// SIMATIC STEP 7 (V5.x) project AEX52
// CPU: CPU
// station: P_ADR_BUS
// station: _S7H_BUSSYSTEM_CT
// station: Matériel
// station: API
// station: P_ADR_BUS
// station: Configuration
// station: MOP
// program: PROG
// program: SAFETY_V2
// program: S120_CU320_2_PN

SYMBOL_TABLE
"ITS0"	DB 1100	FB 1100	// ILOT : DB INSTANCE FB1100
"ITSZ1_AU_ES_FZ"	DB 1110	FB 1110	// Z1 : DB D'INSTANCE DU FB 1110
"ITSZ1SOP"	DB 1111	FB 1111	// Z1 : DB D'INSTANCE DU FB 1111
"ITSZ1SOPR"	DB 1112	FB 1112	// Z1 : DB D'INSTANCE DU FB 1112
"ITSZ1VAR"	DB 1113	FB 1113	// Z1 : DB D'INSTANCE DU FB 1113
"TSM"	DB 1279	DB 1279	// STD - DB global pour la Tâche de Sécurité
"TSE_AMONT"	DB 1286	FB 1692	// STD - INSTANCE DB OF FB 1692 (F_SENDDP) SAFETY DATA SEND
"TSR_AMONT"	DB 1287	FB 1693	// STD - INSTANCE DB OF FB 1693 (F_RCVDP) SAFETY DATA RECEIVE
"TSE_AVAL"	DB 1288	FB 1692	// STD - INSTANCE DB OF FB 1692 (F_SENDDP) SAFETY DATA SEND
"TSR_AVAL"	DB 1289	FB 1693	// STD - INSTANCE DB OF FB 1693 (F_RCVDP) SAFETY DATA RECEIVE
"F_GLOBDB"	DB 1300	DB 1300	// F_: F_Global_Data Block
"F_TON"	FB 185	FB 185	// F_: Timer Switch On Delay
"F_TOF"	FB 186	FB 186	// F_: Timer Switch Off Delay
"TS0"	FB 1100	FB 1100	// ILOT: FB Gestion SAFETY ilot
"TSZ1_AU_ES_FZ"	FB 1110	FB 1110
"TSZ1_SOP"	FB 1111	FB 1111
"TSZ1_SOPR"	FB 1112	FB 1112
"TSZ1_VAR"	FB 1113	FB 1113
"F_SENDDP"	FB 1692	FB 1692	// F_: Send Data via PROFIBUS DP / PROFINET IO
"F_RCVDP"	FB 1693	FB 1693	// F_: Receive Data via PROFIBUS DP / PROFINET IO
"F_ACK_GL"	FB 1695	FB 1695	// Acquittement global de toutes les périphéries F d'un groupe d'exécution F
"BFS_BSEC1"	FB 1710	FB 1710
"BFS_BSECTR1"	FB 1711	FB 1711
"BFS_PORTE1"	FB 1712	FB 1712
"BFS_AIR1"	FB 1713	FB 1713
"BFS_CRM1"	FB 1714	FB 1714
"BFS_CR1"	FB 1715	FB 1715
"BFS_CAME_ROBOT1"	FB 1716	FB 1716
"BFS_MUT1"	FB 1717	FB 1717
"BFS_BIMA1"	FB 1721	FB 1721
"0_00_TSSAFETY"	FC 1100	FC 1100	// STD - FACILITY: EXECUTION F GROUP ASSOCIATE TO OB32 (NORMAL TASK)
"0_00_TSCYCLE"	FC 1101	FC 1101	// CALL OPERATOR NOT IN ZONE FB LINKED IN FACILITY
"P0OP1BAU1"	I 2.0	BOOL	// [P0SB1A.M08]: OPERATOR 1 EGS.CHANNEL 1 / BP ARRET D URGENCE OPERATEUR 1 (VOIE 1)
"P0OP2BAU1"	I 2.1	BOOL	// [P0SB1A.M08]: OPERATOR 2 EGS.CHANNEL 1 / BP ARRET D URGENCE OPERATEUR 2 (VOIE 1)
"P0OP3BAU1"	I 2.2	BOOL	// [P0SB1A.M08]: OPERATOR 3 EGS.CHANNEL 1 / BP ARRET D URGENCE OPERATEUR 3 (VOIE 1)
"P0OP4BAU1"	I 2.3	BOOL	// [P0SB1A.M08]: OPERATOR 4 EGS.CHANNEL 1 / BP ARRET D URGENCE OPERATEUR 4 (VOIE 1)
"P0OP1BAU2"	I 2.4	BOOL	// [P0SB1A.M08]: OPERATOR 1 EGS.CHANNEL 2 / BP ARRET D URGENCE OPERATEUR 1 (VOIE 2)
"P0OP2BAU2"	I 2.5	BOOL	// [P0SB1A.M08]: OPERATOR 2 EGS.CHANNEL 2 / BP ARRET D URGENCE OPERATEUR 2 (VOIE 2)
"P0OP3BAU2"	I 2.6	BOOL	// [P0SB1A.M08]: OPERATOR 3 EGS.CHANNEL 2 / BP ARRET D URGENCE OPERATEUR 3 (VOIE 2)
"P0OP4BAU2"	I 2.7	BOOL	// [P0SB1A.M08]: OPERATOR 4 EGS.CHANNEL 2 / BP ARRET D URGENCE OPERATEUR 4 (VOIE 2)
"P0OP1CPOP1"	I 3.0	BOOL	// [P0SB1A.M09]: LIGHT CURTAIN 1 OR LASER 1 (CH 1) / BARRIERE IMMAT OU SCRUTATEUR
"P0_FDI_RES11"	I 3.1	BOOL	// [P0SB1A.M09]: SPARE SAFE DIGITAL INPUT / RESERVE ENTREE DE SECURITE
"P0OP2CPOP1"	I 3.2	BOOL	// [P0SB1A.M09]: LIGHT CURTAIN 2 OR LASER 2 (CH 1) / BARRIERE IMMAT OU SCRUTATEUR
"P0_FDI_RES21"	I 3.3	BOOL	// [P0SB1A.M09]: SPARE SAFE DIGITAL INPUT / RESERVE ENTREE DE SECURITE
"P0OP1CPOP2"	I 3.4	BOOL	// [P0SB1A.M09]: LIGHT CURTAIN 1 OR LASER 1 (CH 2) / BARRIERE IMMAT OU SCRUTATEUR
"P0_FDI_RES12"	I 3.5	BOOL	// [P0SB1A.M09]: SPARE SAFE DIGITAL INPUT / RESERVE ENTREE DE SECURITE
"P0OP2CPOP2"	I 3.6	BOOL	// [P0SB1A.M09]: LIGHT CURTAIN 2 OR LASER 2 (CH 2) / BARRIERE IMMAT OU SCRUTATEUR
"P0_FDI_RES22"	I 3.7	BOOL	// [P0SB1A.M09]: SPARE SAFE DIGITAL INPUT / RESERVE ENTREE DE SECURITE
"P0OP3CPOP1"	I 4.0	BOOL	// [P0SB1A.M10]: LIGHT CURTAIN 3 (CHANNEL 1)  / BARRIERE IMMATERIELLE (VOIE 1)
"P0_FDI_RES31"	I 4.1	BOOL	// [P0SB1A.M10]: SPARE SAFE DIGITAL INPUT / RESERVE ENTREE DE SECURITE
"P0OP4CPOP1"	I 4.2	BOOL	// [P0SB1A.M10]: LIGHT CURTAIN 4 (CHANNEL 1)  / BARRIERE IMMATERIELLE (VOIE 1)
"P0_FDI_RES41"	I 4.3	BOOL	// [P0SB1A.M10]: SPARE SAFE DIGITAL INPUT / RESERVE ENTREE DE SECURITE
"P0OP3CPOP2"	I 4.4	BOOL	// [P0SB1A.M10]: LIGHT CURTAIN 3 (CHANNEL 2)  / BARRIERE IMMATERIELLE (VOIE 2)
"P0_FDI_RES32"	I 4.5	BOOL	// [P0SB1A.M10]: SPARE SAFE DIGITAL INPUT / RESERVE ENTREE DE SECURITE
"P0OP4CPOP2"	I 4.6	BOOL	// [P0SB1A.M10]: LIGHT CURTAIN 4 (CHANNEL 2)  / BARRIERE IMMATERIELLE (VOIE 2)
"P0_FDI_RES42"	I 4.7	BOOL	// [P0SB1A.M10]: SPARE SAFE DIGITAL INPUT / RESERVE ENTREE DE SECURITE
"Z1CCSC1"	I 10.0	BOOL	// (Z1ZB.M02): SAFETY COMMON CONTROL SC1
"Z1CCES"	I 10.1	BOOL	// (Z1ZB.M02): SAFETY COMMON CONTROL ES
"Z1CCFZ"	I 10.2	BOOL	// (Z1ZB.M02): SAFETY COMMON CONTROL FZ
"Z1CCSC4"	I 10.3	BOOL	// (Z1ZB.M02): SAFETY COMMON CONTROL SC4
"Z1CP7B"	I 11.0	BOOL	// (Z1ZB.M03): 7 BARS PRESSURE CONTROL
"Z1CRM"	I 11.1	BOOL	// (Z1ZB.M03): CHECK GROUND RELAY
"BAUI"	I 13.0	BOOL	// (Z1ZB.M07): FACILITY EMERGENCY STOP
"Z1BAU2"	I 13.1	BOOL	// (Z1ZB.M07): ZONE EMERGENCY STOP
"Z1SSZ"	I 13.2	BOOL	// (Z1ZB.M07): ZONE SAFETY SELECTOR
"Z1CPOP1"	I 19.0	BOOL	// (Z1ZB.M08): LIGHT CURTAIN 1
"Z1CPOP2"	I 19.1	BOOL	// (Z1ZB.M08): LIGHT CURTAIN 2
"Z1RB3CCB24Z"	I 60.4	BOOL	// (Z1RB3.M02): ELECTRICAL CIRCUIT BREAKER 24V (24Z)
"Z1RB3CCB24R"	I 60.5	BOOL	// (Z1RB3.M02): ELECTRICAL CIRCUIT BREAKER 24V (24R)
"Z1SPA1BMCY"	I 100.7	BOOL	// (Z1SPA1.I0): CYCLE START BUTTON
"Z1SPA1BDACY"	I 101.0	BOOL	// (Z1SPA1.I1): CYCLE STOP REQUEST BUTTON
"Z1SPA1SPES"	I 101.3	BOOL	// (Z1SPA1.I1): SWITCH ON / OFF GATE
"Z1SPA1SS"	I 103.7	BOOL	// (Z1SPA1.SI0): SAFETY SELECTOR
"Z1SPA1CFP"	I 104.0	BOOL	// (Z1SPA1.SI1): DOOR CLOSED CONTROL
"P0RBXCFRO_ES"	I 104.6	BOOL	// [P0RBX]: RB OUTPUT - FRO ES COMMON CHECK / CONTROLE FRO MISE EN SERVICE
"P0RBXCFRO_ZF1"	I 104.7	BOOL	// [P0RBX]: RB OUTPUT - FRO FZ1 COMMON CHECK / CONTROLE FRO FERMETURE ZONE 1
"P0RBXCFRO_ZF2"	I 105.0	BOOL	// [P0RBX]: RB OUTPUT - FRO FZ2 COMMON CHECK / CONTROLE FRO FERMETURE ZONE 2
"Z1SPA2BMCY"	I 110.7	BOOL	// (Z1SPA2.I0): CYCLE START BUTTON
"Z1SPA2BDACY"	I 111.0	BOOL	// (Z1SPA2.I1): CYCLE STOP REQUEST BUTTON
"Z1SPA2SPES"	I 111.3	BOOL	// (Z1SPA2.I1): SWITCH ON / OFF GATE
"Z1SPA2SS"	I 113.7	BOOL	// (Z1SPA2.SI0): SAFETY SELECTOR
"Z1SPA2CFP"	I 114.0	BOOL	// (Z1SPA2.SI1): DOOR CLOSED CONTROL
"ZZXCP7B"	I 201.0	BOOL	// [ZZXZB.M03]: CHECK EV 7 BARS
"ZZXCRM"	I 201.1	BOOL	// [ZZXZB.M03]: CHECK GROUND RELAY
"ZZXCCB400_1"	I 201.2	BOOL	// [ZZXZB.M03]: BREAKER CONTROL 400V (SDB1)
"ZZXCRO_11"	I 201.3	BOOL	// [ZZXZB.M03]: SAFETY CONTACTOR CONTROL 1 (SDB1)
"ZZXCRO_12"	I 201.4	BOOL	// [ZZXZB.M03]: SAFETY CONTACTOR CONTROL 2 (SDB1)
"ZZXCCB400_2"	I 201.5	BOOL	// [ZZXZB.M03]: BREAKER CONTROL 400V (SDB2)
"ZZXCRO_21"	I 201.6	BOOL	// [ZZXZB.M03]: SAFETY CONTACTOR CONTROL 1 (SDB2)
"ZZXCRO_22"	I 201.7	BOOL	// [ZZXZB.M03]: SAFETY CONTACTOR CONTROL 2 (SDB2)
"ZZXBAUI1"	I 202.0	BOOL	// [ZZXZB.M06]: EGS FACILITY (MOP/LOP) - CHANNEL 1
"ZZXBAU1"	I 202.1	BOOL	// [ZZXZB.M06]: EGS ZONE (SOP/DLOP) - CHANNEL 1
"ZZXSSZ1"	I 202.2	BOOL	// [ZZXZB.M06]: SAFETY ZONE SELECTOR - CHANNEL 1
"ZZXBAUI2"	I 202.4	BOOL	// [ZZXZB.M06]: EGS FACILITY (MOP/LOP) - CHANNEL 2
"ZZXBAU2"	I 202.5	BOOL	// [ZZXZB.M06]: EGS ZONE (SOP/DLOP) - CHANNEL 2
"ZZXSSZ2"	I 202.6	BOOL	// [ZZXZB.M06]: SAFETY ZONE SELECTOR - CHANNEL 2
"ZZXIFRO1"	I 213.0	BOOL	// [ZZXZB.M08]: FRO1 INTERNAL CHECK
"ZZXIFRO2"	I 214.0	BOOL	// [ZZXZB.M09]: FRO2 INTERNAL CHECK
"P0OPXBP11"	I 339.0	BOOL	// [P0SB1A.M09]: OPX T-STAND BUTTON 1 - CHANNEL 1 / BIMANUEL X BOUTON 1 (VOIE 1)
"P0OPXBP21"	I 339.1	BOOL	// [P0SB1A.M09]: OPX T-STAND BUTTON 2 - CHANNEL 1 / BIMANUEL X BOUTON 2 (VOIE 1)
"P0OPXBP12"	I 339.4	BOOL	// [P0SB1A.M09]: OPX T-STAND BUTTON 1 - CHANNEL 2 / BIMANUEL X BOUTON 1 (VOIE 2)
"P0OPXBP22"	I 339.5	BOOL	// [P0SB1A.M09]: OPX T-STAND BUTTON 2 - CHANNEL 2 / BIMANUEL X BOUTON 2 (VOIE 2)
"BA0"	M 0.0	BOOL	// FACILITY: BIT ALWAYS OFF
"BA1"	M 0.1	BOOL	// FACILITY: BIT ALWAYS ON
"BA1LIEN"	M 0.2	BOOL	// FACILITY: BIT ALWAYS ON (LINK IN THE PROGRAMMING NETWORK)
"SHUNT"	M 0.3	BOOL	// FACILITY: BIT  FOR BYPASS SOME FUNCTIONS DURING THE TEST
"PERSO"	M 0.4	BOOL	// NEED TO PERSONALIZE BY THE PROGRAMMER
"POUB"	M 0.5	BOOL	// BIT TRASH
"SYSFROID"	M 0.7	BOOL	// DETECTING COLD START PLC (OB102)
"DEF_MAJ"	M 10.0	BOOL	// FACILITY: MAJOR FAULT (SAFETY)
"IADF"	M 10.1	BOOL	// FACILITY: FAULT RESET INFORMATION (SAFETY)
"IR"	M 10.2	BOOL	// FACILITY: CONTROL ON INFORMATION (SAFETY)
"P0OP1CRSP0"	M 12.0	BOOL	// P0: SAFETY RESET CONDITION / CONDITION DE REARMEMENT SECURITE
"P0OP2CRSP0"	M 12.1	BOOL	// P0: SAFETY RESET CONDITION / CONDITION DE REARMEMENT SECURITE
"Z1DEF_MAJ"	M 100.0	BOOL	// ZONE 1: MAJOR FAULT (SAFETY)
"Z1IADF"	M 100.1	BOOL	// ZONE 1: FAULT RESET INFORMATION (SAFETY)
"Z1IR"	M 100.2	BOOL	// ZONE 1: CONTROL ON INFORMATION (SAFETY)
"Z1IAFJ"	M 100.3	BOOL	// ZONE 1: END OF PRODUCTION STOP INFORMATION (SAFETY)
"P0OPXCRSP0"	M 103.2	BOOL	// P0OPX: SAFETY RESET CONDITION / CONDITION DE REARMEMENT SECURITE
"ZZXDEF_MAJ"	M 200.0	BOOL	// ZONE ZX: MAJOR FAULT (SAFETY)
"ZZXIADF"	M 200.1	BOOL	// ZONE ZX: FAULT RESET INFORMATION (SAFETY)
"ZZXIR"	M 200.2	BOOL	// ZONE ZX: CONTROL ON INFORMATION (SAFETY)
"ZZXIAFJ"	M 200.3	BOOL	// ZONE ZX: END OF PRODUCTION STOP INFORMATION (SAFETY)
"P0IAVARR"	M 201.0	BOOL	// P0: INFORMATION INVERTER STOP / INFO ARRET IMMEDIAT VARIATEUR
"P0_AT_P0OPX"	M 204.0	BOOL	// P0: OPERATOR P0OPX WORK AUTORIZATION / AUTORISATION DE TRAVAIL OPERATEUR P0OPX
"P0_ET_P0OPX"	M 204.1	BOOL	// P0: OPERATOR P0OPX WORK RECORD / ENREGISTREMENT TRAVAIL OPERATEUR P0OPX
"Z1RCM"	Q 10.7	BOOL	// (Z1ZB.M05): CHECK GROUND RELAY
"Z1RSC1"	Q 25.0	BOOL	// (Z1ZB.M09): SAFETY COMMON RELAY SC1
"Z1RES"	Q 25.1	BOOL	// (Z1ZB.M09): SAFETY COMMON RELAY ES
"Z1RFZ"	Q 25.2	BOOL	// (Z1ZB.M09): SAFETY COMMON RELAY FZ
"Z1RSC4"	Q 25.3	BOOL	// (Z1ZB.M09): SAFETY COMMON RELAY SC4
"DPRD_DAT"	SFC 14	SFC 14	// Read Consistent Data of a Standard DP Slave
"DPWR_DAT"	SFC 15	SFC 15	// Write Consistent Data to a Standard DP Slave
"STP"	SFC 46	SFC 46	// Change the CPU to STOP
END_SYMBOL_TABLE

// FB 185: know-how protected block, not included

// FB 186: know-how protected block, not included

FUNCTION_BLOCK "TS0"	// FB 1100
VERSION : 0.3
VAR
  ACK_GLB : FB 1695;	//FACILITY: GLOBAL FAULT RESET FOR SAFETY MODULE/AQUIT GENERAL DEF MATERIEL SAFET
  Z1CRM : FB 1714;	//Z1: GROUND RELAY CHECK / CONTROLE RELAI DE MASSE
END_VAR
BEGIN
// body was compiled from another editor; compiled code not shown
END_FUNCTION_BLOCK

FUNCTION_BLOCK "TSZ1_AU_ES_FZ"	// FB 1110
VERSION : 0.3
VAR
  Z1AU : FB 1710;	//Z1: EMERGENCY STOP RELAY CONTROL / GESTION BOUCLE DE SECURITE AU
  Z1ES : FB 1710;	//Z1: POWER ON RELAY CONTROL / GESTION RELAY MISE EN SERVICE
  Z1FZ : FB 1710;	//Z1: CLOSED ZONE SAFETY LOOP MANAGEMENT / GESTION BOUCLE DE SECURITE FZ
  Z1AIR : FB 1713;	//Z1: PRESSURIZING VALVE CONTROL / GESTION ELECTROVANNE DE MISE EN AIR
  Z1PORTE1 : FB 1712;	//Z1: DOOR 1 CONTROL / GESTION PORTE 1
  Z1PORTE2 : FB 1712;	//Z1: DOOR 2 CONTROL / GESTION PORTE 2
END_VAR
VAR_TEMP
  X1IBFF : BOOL ;	//AUX1 SAFETY CIRCUIT CORRECT WORKING INFORMATION / AUX BON FONCTIONNEMENT FILERI
  X2IBFF : BOOL ;	//AUX2 SAFETY CIRCUIT CORRECT WORKING INFORMATION / AUX BON FONCTIONNEMENT FILERI
  X3IBFF : BOOL ;	//AUX3 SAFETY CIRCUIT CORRECT WORKING INFORMATION / AUX BON FONCTIONNEMENT FILERI
  X1AUCAR : BOOL ;	//AUX1 CONDITIONS WITH RESET EMERGENCY STOP / AUX CONDITION AVEC REARMEMENT AU
  X2AUCAR : BOOL ;	//AUX2 CONDITIONS WITH RESET EMERGENCY STOP / AUX CONDITION AVEC REARMEMENT AU
  X1ESCAR : BOOL ;	//AUX1 CONDITIONS WITH RESET POWER ON / AUX1 CONDITIONS AVEC REARMEMENT EN SERVIC
  X2ESCAR : BOOL ;	//AUX2 CONDITIONS WITH RESET POWER ON / AUX2 CONDITIONS AVEC REARMEMENT EN SERVIC
END_VAR
BEGIN
// body was compiled from another editor; compiled code not shown
END_FUNCTION_BLOCK

FUNCTION_BLOCK "TSZ1_SOP"	// FB 1111
TITLE = POWER ON RELAY CONTROL
VERSION : 0.2
VAR
  C0SOP : FB 1710;
  F0SOP : FB 1710;
  G0SOP : FB 1710;
  P0SOP : FB 1710;
  P01SOP : FB 1710;
  P01SOP_Secu : BOOL ;	//Activation boucle de sécurité opérateur
  P02SOP : FB 1710;
  P02SOP_Secu : BOOL ;	//Activation boucle de sécurité opérateur
  F1BIMA : FB 1719;
  F2BIMA : FB 1719;
  F3BIMA : FB 1719;
END_VAR
VAR_TEMP
  C0SOP_Car : BOOL ;
  C0SOP_Csr : BOOL ;
  G0SOP_Car : BOOL ;
  G0SOP_Csr : BOOL ;
  P0SOP_Car : BOOL ;
  P0SOP_Csr : BOOL ;
  P01SOP_Car : BOOL ;
  P01SOP_Csr : BOOL ;
  P02SOP_Car : BOOL ;
  P02SOP_Csr : BOOL ;
  F0SOP_Car : BOOL ;
  F0SOP_Csr : BOOL ;
  C0SOP_csecu0 : BOOL ;
  C0SOP_csecu1 : BOOL ;
  F0SOP_csecu0 : BOOL ;
  F0SOP_csecu1 : BOOL ;
  G0SOP_csecu0 : BOOL ;
  G0SOP_csecu1 : BOOL ;
  P0SOP_csecu0 : BOOL ;
  P0SOP_csecu1 : BOOL ;
  P01SOP_csecu0 : BOOL ;
  P01SOP_csecu1 : BOOL ;
  P02SOP_csecu0 : BOOL ;
  P02SOP_csecu1 : BOOL ;
END_VAR
BEGIN
// body was compiled from another editor; compiled code not shown
END_FUNCTION_BLOCK

FUNCTION_BLOCK "TSZ1_SOPR"	// FB 1112
TITLE = CLOSED ZONE ELECTRICAL COMMON MANAGEMENT (FZ)
//GESTION DU COMMUN ELECTRIQUE : FERMETURE ZONE (FZ)
VERSION : 0.2
VAR
  R1CAME : FB 1716;
  R1SOPR : FB 1710;
END_VAR
VAR_TEMP
  R1SOPR_Car : BOOL ;	//R1 Conditions avec réarmement
  R1SOPR_Csr : BOOL ;	//R1 Conditions sans réarmement
  R1SOPR_csecu0 : BOOL ;
  R1SOPR_csecu1 : BOOL ;
END_VAR
BEGIN
// body was compiled from another editor; compiled code not shown
END_FUNCTION_BLOCK

FUNCTION_BLOCK "TSZ1_VAR"	// FB 1113
VERSION : 0.2
VAR
  Z1FZTR : FB 1711;	//Z1: CLOSED ZONE TEMPO SAFETY LOOP MANAGEMENT / GESTION BOUCLE SECURITE FZTR
END_VAR
BEGIN
// body was compiled from another editor; compiled code not shown
END_FUNCTION_BLOCK

// FB 1692: know-how protected block, not included

// FB 1693: know-how protected block, not included

// FB 1695: know-how protected block, not included

FUNCTION_BLOCK "BFS_BSEC1"	// FB 1710
//**********************************************************************
//*                             BFS_BSEC1                               *
//**********************************************************************
//(in english further below)
//DESCRIPTION: 
//************ 
//Le FB1710 "BFS_BSEC1" est un relais de securite logiciel programme en Step7 + 
//Distributed Safety pour assurer la surete de fonctionnement d'une boucle de 
//securite geree par automate Simatic Failsafe.
//C'est une evolution de la BFS_BSEC pour le Scube Safety V2
//
//Son role est 
//"De piloter une sortie F-DO ou PME-F, sur laquelle est cablee en fonction 
//du besoin process, un contacteur pour les energies de puissance 
//securisees et/ou un relais pour les communs de commande 24V et/ou une 
//electrovanne pour les energies de puissance pneumatiques. 
//"De controler la coherence entre le pilotage et l'etat des retours
//"De mettre a disposition du programme standard un commun de securite " 
//soft " pour conditionner le pilotage des sorties automates des mouvements a la 
//presence effective des communs de commande 24V et/ou des energies de puissance 
//et aussi pour conditionner les communs en aval (effet cascade)
//"D'avertir du mauvais fonctionnement de la boucle de securite (Alarme : 
//pas de retour alors que la sortie est pilotee, Defaut : retour present alors 
//que la sortie n'est pas pilotee)
//
//Le FB prend en compte les informations necessaires a la securisation de la 
//boucle de securite concernee.
//Il renseigne sur l'etat de defaillance de la fonction de securite.
//
//Les blocs associes pour le diagnostic via IHMP+ sont :
//BF_IHMCR1 pour les fonctions AU, ES, ZF et toute autre utilisation du 
//BFS_BSEC1 par exemple SOP …
//Le bloc BFS_BSEC1 peut egalement etre utilise pour la gestion du RL (Relais de 
//ligne) des fonctions variateurs Scube (Attention dans ce cas le diagnostic, pour 
//IHMP+, est realise par la BF associee a la fonction variateur)
//
//
//*************************English Information*******************************
//Description
//***********
//The FB1710 "BFS_BSEC1" is a software safety relay in Step 7 + Distributed 
//Safety to ensure the dependability of a safety loop managed by a Simatic 
//Failsafe PLC.
//It's an evolution of the BFS_BSEC with the Safety Scube V2.
//
//It serves: 
//"to control an F-DO or PME-F output, to which a contactor for the 
//safe power supplies and/or an relay for the safe commons 24V and/or a solenoid 
//valve for the safe power pneumatic fluid is/are wired according to process 
//requirements.
//"to check the consistency between the control and the status of the 
//feedbacks
//"to make a "software" safe common 24 V available to the standard program, to 
//make the control of PLC movement outputs conditional on the effective presence 
//of 24V control commons and/or power supplies and also to make the downstream 
//commons 24 V conditional (daisy-chained effect)
//"to give the alert in the event of incorrect operation of the safety loop 
//(Alarm: no feedback although the output is controlled, Fault: feedback present 
//although the output is not controlled)
//
//The FB takes into account the Data required to secure the safety loop concerned.
//It gives details on the failure status of the safety function and updates the 
//data from lien_sec used in the standard program.
//
//The associated blocks for the diagnostics via IHMP+ are:
//BF_IHMCR1 for the functions AU, ES, ZF and any other use of BFS_BSEC1 for 
//example SOP …
//The block BFS_BSEC1 can also be used to manage the RL (Line relay)of the Scube 
//drive functions (Attention in this case the diagnosis, for IHMP+, is carried out 
//with the BF associated with the drive function. 
//
AUTHOR : SIEMENS
FAMILY : RENAULT
NAME : BSEC1
VERSION : 1.0
VAR_INPUT
  Ibff : BOOL ;	//Safety circuit correct working info./Information bon fonctionnement filerie
  Car : BOOL ;	//Conditions with control on/Conditions avec rearmement
  Csr : BOOL ;	//Conditions without control on/Conditions sans rearmement
  CSecu0 : BOOL ;	//Feedbacks check without control/Controle Retours sans pilotage
  CSecu1 : BOOL ;	//Feedbacks check with control/Controle Retours avec Pilotage
  Iadf : BOOL ;	//Fault reset/Annulation defaut
  Ir : BOOL ;	//Function control on/Rearmement fonction
END_VAR
VAR_OUTPUT
  DO_F : BOOL ;	//F-DO output control/Commande sortie F-DO
  Secu : BOOL ;	//Similar with DO-F/Identique a DO_F
  Secu_OK : BOOL ;	//Safety loop correct/Boucle de securite valide
  Def : BOOL ;	//Discrepancy fault in the deactivation/Defaut de discordance a la desactivation
END_VAR
VAR
  x : BOOL  := TRUE;	//Bit of instance location/Bit de localisation de l'instance
  IHMDef : BOOL ;	//Discrepancy fault in the deactivation/Defaut de discordance a la desactivation
  IHMAla : BOOL ;	//Discrepancy fault in the activation/Def de discordance a l'activation (Ala)
  xSecu : BOOL ;	//Auxiliary bit/Bit auxiliaire
  M_ala : BOOL ;	//Alarm memory/Memoire alarme
  M_ar : BOOL ;	//Car memory (cond with Ctrl On)/Memoire car
  xIr : BOOL ;	//Auxiliary bit control on/Bit auxiliaire rearmement
  TON_Disc : FB 185;	//Discrepancy detection timer/Tempo de detection discordance
END_VAR
VAR_TEMP
  FP_Ir : BOOL ;	//Rising edge bit Ir (Control on information)/Bit front montant Ir
END_VAR
BEGIN
// body was compiled from another editor; compiled code not shown
END_FUNCTION_BLOCK

FUNCTION_BLOCK "BFS_BSECTR1"	// FB 1711
//**********************************************************************
//*                            BFS_BSECTR1                              *
//**********************************************************************
//(in english further below)
//DESCRIPTION: 
//************ 
//Le FB1711 "BFS_BSECTR1" est un relais de securite logiciel temporise a la 
//retombee programme en Step7 + Distributed Safety pour assurer la surete de 
//fonctionnement d'une boucle de securite gere par automate Simatic Failsafe.
//C'est une evolution de la BFS_BSECTR pour le Scube Safety V2
//
//Son role est 
//"De piloter une sortie F-DO ou PME-F temporise a la retombee, sur 
//laquelle est cablee en fonction du besoin process, un contacteur
//pour les energies de puissance securisees et/ou un relais pour 
//les communs de commande 24V securises.
//"De controler la coherence entre le pilotage et l'etat des retours
//"De mettre a disposition du programme standard un commun de securite " 
//soft " pour conditionner le pilotage des sorties automates des mouvements a la 
//presence effective des communs de commande 24V et/ou des energies de puissance
//"D'avertir du mauvais fonctionnement de la boucle de securite (Alarme : 
//pas de retour alors que la sortie est pilotee, Defaut : retour present alors 
//que la sortie n'est pas pilotee)
//
//Le FB prend en compte les informations necessaires a la securisation de la 
//boucle de securite concernee.
//
//Il renseigne sur l'etat de defaillance de la fonction de securite. 
//
//Les blocs associes pour le diagnostic via IHMP+ sont :
//BF_IHMCR1 pour la fonction ESTR ou toutes les autres utilisation du 
//BFS_BSECTR1
//
//*************************English Information*******************************
//Description
//***********
//The FB1711 "BFS_BSECTR" is a software safety relay with a delay when 
//falling, programmed in Step 7 + Distributed Safety to ensure the dependability 
//of a safety loop managed by a Simatic Failsafe PLC.
//It's an evolution of the BFS_BSEC with the Safety Scube V2.
//
//It serves: 
//"to control an F-DO or PME-F output with a deactivation delay, to which a 
//contactor for the safe power supplies and/or a relay for the safe commons 24V 
//is/are wired according to process requirements.
//"to check the consistency between the control and the status of the feedbacks
//"to make a "software" safe common 24 V available to the standard program, to 
//make the control of PLC movement outputs conditional on the effective presence 
//of 24V control commons and/or power supplies. 
//"to give the alert in the event of incorrect operation of the safety loop 
//(Alarm: no feedback although the output is controlled, Fault: feedback present 
//although the output is not controlled)
//
//The FB takes account of the Data required to secure the safety loop concerned.
//It gives details on the failure status of the safety function.
//
//The associated blocks for the diagnostics via IHMP+ are:
//BF_IHMCR1 for the ESTR function or all other uses of BFS_BSECTR1 
//BF_FONC_VAR_S for the RL function of FONC_VAR
AUTHOR : SIEMENS
FAMILY : RENAULT
NAME : BSECTR1
VERSION : 1.0
VAR_INPUT
  DSecu : BOOL ;	//Safety dependence/Dependance securite
  Cci : BOOL ;	//Immediate cut-off conditions/Conditions coupure immediate
  CSecu0 : BOOL ;	//Feedbacks check without control/Controle Retours sans pilotage
  CSecu1 : BOOL ;	//Feedbacks check with control/Controle Retours avec Pilotage
  Iadf : BOOL ;	//Fault reset/Annulation defaut
  Ir : BOOL ;	//Function control on/Rearmement fonction
  Tps_secu : TIME ;	//Relay deactivating time(Max.=2s)/Temps de retombee du relais (Maxi 2s
END_VAR
VAR_OUTPUT
  DO_F : BOOL ;	//F-DO output control/Commande sortie F-DO
  Secu : BOOL ;	//Similar with DO-F/Identique à DO_F
  Secu_OK : BOOL ;	//Safety loop correct/Boucle de securite valide
  Def : BOOL ;	//Discrepancy fault in the deactivation/Défaut de discordance à la desactivation
END_VAR
VAR
  x : BOOL ;	//Bit of instance location/Bit de localisation de l'instance
  IHMDef : BOOL ;	//Discrepancy fault in the deactivation/Defaut de discordance a la desactivation
  IHMAla : BOOL ;	//Discrepancy fault in the activation/Def de discordance a l'activation (Ala)
  xSecu : BOOL ;	//Auxiliary bit/Bit auxiliaire
  M_ala : BOOL ;	//Alarm memory/Memoire alarme
  M_Cci : BOOL ;	//Cci memory / memoire Cci
  xIr : BOOL ;	//Auxiliary bit control on/Bit auxiliaire rearmement
  TON_Disc : FB 185;	//Discrepancy detection timer/Tempo de detection discordance
  TOFF_Max : FB 186;	//Timer of relay deactivation with 2s max./Tempo de retombee relais avec 2 s max
  TOFF_Secu : FB 186;	//Timer of relay deactivation/Tempo de retombee relais
END_VAR
VAR_TEMP
  FP_Ir : BOOL ;	//Rising edge bit Ir (Control on information)/Bit front montant Ir
END_VAR
BEGIN
// body was compiled from another editor; compiled code not shown
END_FUNCTION_BLOCK

FUNCTION_BLOCK "BFS_PORTE1"	// FB 1712
//**********************************************************************
//*                             BFS_PORTE1                              *
//**********************************************************************
//(in english further below)
//DESCRIPTION: 
//************ 
//Le FB1712 "BFS_PORTE1" est un relais de securite logiciel programme en Step7 + 
//Distributed Safety.
//C'est une evolution de la BFS_PORTE pour le Scube Safety V2
//
//Ce FB assure la gestion des composants associes a une porte d'acces Zone.
//Il fournit les conditions pour l'activation des boucles de securité ES et ZF.
//Il controle le respect de la procedure d'intervention dans la zone.
//Il controle le bon fonctionnement de la gache, desactivation de 
//l'information cfp a chaque ouverture d'un des deux commutateurs SS ou SPES.
//
//Le blocs associe pour le diagnostic via IHMP+ est:
//BF_IHMPORTE1
//
//*************************English Information*******************************
//Description
//***********
//The FB1712 "BFS_BSEC1" is a software safety relay in Step 7 + Distributed 
//Safety. 
//It's an evolution of the BFS_PORTE with the Safety Scube V2.
//
//This FB ensures the management of components combined with a access gate into 
//an 
//area.
//It gives the conditions for the activation of safety loops ES and ZF. 
//It checks the respect of the intervention procedure in the area.
//It checks the correct working of the striker, deactivation of information cfp 
//in every opening of one of both switches SS or SPES.
//
//The associated block for the diagnostic via IHMP+ is:
//BF_IHMPORTE1 
AUTHOR : SIEMENS
FAMILY : RENAULT
NAME : PORTE1
VERSION : 1.0
VAR_INPUT
  Ss : BOOL ;	//Safety selector/Selecteur de Securite
  Cfp : BOOL ;	//Door closing check/Controle Fermeture Portillon
  Spes : BOOL ;	//Door enable selector/Selecteur Portillon En Service
  Iadf : BOOL ;	//Fault reset/Acquittement
END_VAR
VAR_OUTPUT
  ES_Car : BOOL ;	//Door validated for ES/Porte Ok pour ES
  FZ_Car : BOOL ;	//Door validated for FZ/Porte Ok pour FZ
END_VAR
VAR
  x : BOOL ;	//Bit of instance location/Bit de localisation de l'instance
  DPI : BOOL ;	//Maintenance procedure fault/Defaut procedure d'intervention
  DemOuv : BOOL ;	//Request for door opening/Demande ouvertrure porte
  XSel : BOOL ;	//Edge auxiliary/Auxilliaire de front
END_VAR
BEGIN
// body was compiled from another editor; compiled code not shown
END_FUNCTION_BLOCK

FUNCTION_BLOCK "BFS_AIR1"	// FB 1713
//**********************************************************************
//*                             BFS_AIR1                                *
//**********************************************************************
//(in english further below)
//DESCRIPTION: 
//************ 
//Le FB1713 assure la gestion d'un panneau pneumatique pour une zone. Il peut 
//piloter les electrovannes 7 bars de mise en pression progressive et de shunt de 
//mise en pression progressive.
//C'est une evolution de la BFS_BSECTR pour le Scube Safety V2
// 
//Attention ce pilotage peut egalement etre realise par la sortie securisee de la 
//boucle ES.
//Le FB genere des defauts en cas de dysfonctionnement (incoherence entre le 
//pilotage des electrovannes et le controle de pression pneumatique).
//Ce FB est prevu pour etre utilise avec un panneau classique, comportant les 
//commandes d'une electrovanne de mise en pression progressive et une 
//electrovanne de shunt de mise en pression progressive et un controle de 
//pression.
//Mais il peut egalement etre utilise pour un panneau comportant uniquement  les 
//commandes d'une electrovanne de ligne 7 bars et d'un controle de pression. Dans 
//ce cas, on utilisera la sortie EVMPP pour la commande de l'electrovanne.
//
//Le bloc associe pour le diagnostic via IHMP+ est :
//BF_IHMAIR1
//
//*************************English Information*******************************
//Description
//***********
//The FB1713 manages a zone's air panel. It can control the line solenoid valves 
//(7 Bar) of gradual pressurising and gradual pressurising shunt.
//It's an evolution of the BFS_AIR with the Safety Scube V2. 
//
//Note that this control can also be performed by the In Service loop secured 
//output.
//The FB generates faults if a malfunction occurs (discrepancy between the 
//solenoid valve controls and the air pressure check).
//This FB is designed to be used with a standard panel, including a gradual 
//pressurising solenoid valve, a gradual pressuring shunt solenoid valve and an 
//air pressure check.
//It can also be used for a panel that only has a line solenoid valve (7 bar) and 
//an air pressure check. In this case, we use the EVMPP output for the solenoid 
//valve control.
//
//The associated block for the diagnostic via IHMP+ is:
//BF_IHMAIR1
//
AUTHOR : SIEMENS
FAMILY : RENAULT
NAME : AIR1
VERSION : 1.0
VAR_INPUT
  DSecu : BOOL ;	//Safety dependence/Dependance securite
  Cpa7B : BOOL ;	//Air pressure 7 bars check/Controle Pression Air 7 bars
  Iadf : BOOL ;	//Fault reset/Annulation defaut
  Ir : BOOL ;	//Function control on/Rearmement fonction
  Vptmpp : TIME ;	//Setting value of gradual pressure timer/Val.Paramet.Tempo Mise en Pres. Progr.
END_VAR
VAR_OUTPUT
  EvMPP : BOOL ;	//EV Gradual pressurising valve/EV mise en pression progressive
  ShEvMPP : BOOL ;	//Shunt EV Gradual pressurising valve/Shunt EV mise en pression progressive
  Secu_Ok : BOOL ;	//Pressure air OK/Air Ok
  Def : BOOL ;	//Air fault/Defaut air
END_VAR
VAR
  x : BOOL ;	//Bit of instance location/Bit de localisation de l'instance
  IHMAla : BOOL ;	//Air pressure alarm/Alarme air
  IHMDef : BOOL ;	//Air pressure fault / Defaut Air
  MppT : BOOL ;	//Gradual pressurising time elapsed/Mise en Pression progressive terminee
  Mcp7b : BOOL ;	//Air pressure check memory/Memoire controle pression air
  M_ala : BOOL ;	//Alarm memory/ Memoire alarme
  xIr : BOOL ;	//Auxiliary bit control on/Bit auxiliaire rearmement
  TON_Mpp : FB 185;	//Gradual pressurising timer/Tempo mise en pression progressive
  TON_Disc : FB 185;	//Air fault detection timer/Tempo detection defaut air
END_VAR
VAR_TEMP
  FP_Ir : BOOL ;	//Rising edge bit Ir (Control on information)/Bit front montant Ir
END_VAR
BEGIN
// body was compiled from another editor; compiled code not shown
END_FUNCTION_BLOCK

FUNCTION_BLOCK "BFS_CRM1"	// FB 1714
//**********************************************************************
//*                               BFS_CRM1                              *
//**********************************************************************
//(in english further below)
//DESCRIPTION: 
//************ 
//Le FB1714 "BFS_CRM1" est un relais de securite logiciel programme en Step7 + 
//Distributed Safety.
//Il controle l'etat du relais de controle de masse .
//C'est une evolution de la BFS_CRM pour le Scube Safety V2
//
//Il est a appeler autant de fois qu'il y a d'alimentation 24V.
//Le bloc associe pour le diagnostic via IHMP+ est :
//BF_IHMCRM1
//
//*************************English Information*******************************
//Description
//***********
//The "BFS_CRM1" FB1714 is a software safety relay programmed in Step 7 + 
//Distributed Safety.
//It checks the status of the earthing check relay.
//It's an evolution of the BFS_CRM with the Safety Scube V2.
//
//It is to be integrated for each 24V control power supply.
//The associated block for the diagnostic via IHMP+ is:
//BF_IHMCRM1
AUTHOR : SIEMENS
FAMILY : RENAULT
NAME : CRM1
VERSION : 1.0
VAR_INPUT
  DSecu : BOOL ;	//Safety dependence/Dependance securite
  CSecu : BOOL ;	//Relay feedback information/Information de retour du relais
  Iadf : BOOL ;	//Fault reset/Annulation defaut
END_VAR
VAR_OUTPUT
  Def : BOOL ;	//CRM fault/Defaut CRM
END_VAR
VAR
  x : BOOL ;	//Bit of instance location/Bit de localisation de l'instance
  IHMDef : BOOL ;	//Fault in the deactivation/Defaut a la retombee
  IHMAla : BOOL ;	//Fault in the activation/Defaut a la montee
  xSecu : BOOL ;	//Auxiliary bit/Bit auxiliaire
  Ton_Rsecu : FB 185;	//Timer of discrepancy detection/Tempo de detection discordance
END_VAR
BEGIN
// body was compiled from another editor; compiled code not shown
END_FUNCTION_BLOCK

FUNCTION_BLOCK "BFS_CR1"	// FB 1715
//**********************************************************************
//*                               BFS_CR1                               *
//**********************************************************************
//(in english further below)
//DESCRIPTION: 
//************ 
//Le FB1715 "BFS_CR1" est un relais de securite logiciel programme en Step7 + 
//Distributed Safety.
//C'est une evolution de la BFS_CR pour le Scube Safety V2
//
//Il verifie la coherence entre la commande d'un relais et son etat. 
//
//Le bloc associe pour le diagnostic via IHMP+ est :
//BF_IHMCR1
//
//*************************English Information*******************************
//Description
//***********
//The "BFS_CR1" FB1715 is a software safety relay programmed in Step 7 + 
//Distributed Safety.
//It's an evolution of the BFS_CR with the Safety Scube V2.
//
//It checks the consistency between the relay control and its state.
//
//The associated block for the diagnostic via IHMP+ is:
//BF_IHMCR1
AUTHOR : SIEMENS
FAMILY : RENAULT
NAME : CR1
VERSION : 1.0
VAR_INPUT
  DSecu : BOOL ;	//Conditions with control on/Conditions avec rearmement
  CSecu0 : BOOL ;	//Feedbacks check without control/Controle Retours sans pilotage
  CSecu1 : BOOL ;	//Feedbacks check with control/Controle Retours avec Pilotage
  Iadf : BOOL ;	//Fault reset/Annulation defaut
  Ir : BOOL ;	//Function control on/Rearmement fonction
END_VAR
VAR_OUTPUT
  Secu_OK : BOOL ;	//Secured relay correct/Relais securise valide
  Def : BOOL ;	//Discrepancy fault in the deactivation/Defaut de discordance a la desactivation
END_VAR
VAR
  x : BOOL ;	//Bit of instance location/Bit de localisation de l'instance
  IHMDef : BOOL ;	//Discrepancy fault in the deactivation/Defaut de discordance a la desactivation
  IHMAla : BOOL ;	//Discrepancy fault in the activation/Def de discordance a l'activation (Ala)
  xDsecu : BOOL ;	//Auxiliary bit/Bit auxiliaire
  M_Err : BOOL ;	//Alarm or Fault memory/Memoire alarme ou Defaut
  xIr : BOOL ;	//Auxiliary bit control on/Bit auxiliaire rearmement
  TON_Disc : FB 185;	//Discrepancy detection timer/Tempo de detection discordance
END_VAR
VAR_TEMP
  FP_Ir : BOOL ;	//Rising edge bit Ir (Control on information)/Bit front montant Ir
END_VAR
BEGIN
// body was compiled from another editor; compiled code not shown
END_FUNCTION_BLOCK

FUNCTION_BLOCK "BFS_CAME_ROBOT1"	// FB 1716
//**********************************************************************
//*                               BFS_CAME_ROBOT1                       *
//**********************************************************************
//(in english further below)
//DESCRIPTION: 
//************ 
//Le FB1716 "BFS_CAME_ROBOT1"  est un relais de securite logiciel programme en 
//Step7 + Distributed Safety.
//C'est une evolution de la BFS_CAME_ROBOT pour le Scube Safety V2
//
//Il controle le bon fonctionnement de la came robot (controle came a 0 et 
//controle came a 1 dans un cycle piece).
//Il est a integrer autant de fois qu'il y a de came robot.
//Le bloc associe pour le diagnostic via IHMP+ est :
//BF_IHMCAME_ROBOT1
//
//*************************English Information*******************************
//Description
//***********
//The "BFS_CAME_ROBOT1" FB1716 is a software safety relay in Step 7 + Distributed 
//Safety.
//It's an evolution of the CAME_ROBOT with the Safety Scube V2.  
//
//It checks the correct operation of the Robot cam (cam check set to 0 and cam 
//check set to 1 in a part cycle).
//It should be integrated for each robot cam.
//The associated block for the diagnostic via IHMP+ is:
//BF_IHMCAME_ROBOT1
AUTHOR : SIEMENS
FAMILY : RENAULT
NAME : CAME_RO1
VERSION : 1.0
VAR_INPUT
  Val_Ctrl : BOOL ;	//Check validating/Validation controle
  Came : BOOL ;	//Cam F Input/Entree F came
  C_Came0 : BOOL ;	//Checking Cam at 0 /Controle came à 0
  C_Came1 : BOOL ;	//Checking Cam at 1 /Controle came à 1
  Iadf : BOOL ;	//Fault reset/Annulation defaut
END_VAR
VAR_OUTPUT
  Def : BOOL ;	//Cam fault/Defaut Came
END_VAR
VAR
  x : BOOL ;	//Bit of instance location/Bit de localisation de l'instance
END_VAR
BEGIN
// body was compiled from another editor; compiled code not shown
END_FUNCTION_BLOCK

FUNCTION_BLOCK "BFS_MUT1"	// FB 1717
TITLE = BFS_MUT1
//**********************************************************************
//*                              BFS_MUT1                               *
//**********************************************************************
//(in english further below)
//DESCRIPTION: 
//************ 
//Le FB1717 "BFS_MUT1" assure le fonction de muting d'une barriere anti-intrusion 
//lors d'un passage de caisse.
//C'est une evolution de la BFS_MUT pour le Scube Safety V2
//
//La condition de Muting doit OBLIGATOIREMENT etre une information active pendant 
//tout le deplacement de la charge (memoire de transit).
//
//Les blocs associes pour le diagnostic via IHMP+ sont :
//BF_IHMMUT1 
//
//*************************English Information*******************************
//Description
//***********
//The FB1717 "BFS_MUT1" ensures the muting function of an anti-intrusion barrier 
//during the body's transit.
//It's an evolution of the BFS_MUT with the Safety Scube V2.
//
//The muting condition must be OBLIGATORILY an active information during all the 
//load's transit (transit memory).
//
//The associated block for the diagnostic via IHMP+ is:
//BF_IHMMUT1 
AUTHOR : SIEMENS
FAMILY : RENAULT
NAME : MUTING
VERSION : 1.0
VAR_INPUT
  CAINT1 : BOOL ;	//Anti-intrusion sensor 1/Controle anti-intrusion 1
  CAINT2 : BOOL ;	//Anti-intrusion sensor 2/Controle anti-intrusion 2
  DPAS1 : BOOL ;	//Crossing sensor 1/Detecteur de passage 1
  DPAS2 : BOOL ;	//Crossing sensor 2/Detecteur de passage 2
  CMUT : BOOL ;	//Muting condition/Condition de muting
  Iadf : BOOL ;	//Fault cancellation/Annulation defaut
END_VAR
VAR_OUTPUT
  VMut : BOOL ;	//Active muting warning lamp/Voyant muting actif
  Def : BOOL ;	//Fault/Defaut
END_VAR
VAR
  x : BOOL ;
  IHMDef : BOOL ;	//Fault for the HMI/Defaut pour IHM
  MP0_AINT1 : BOOL ;	//Anti-intrusion sensor 1 temp. reset memory/Mem.passage 0 ctl anti-intrusion 1
  MP0_AINT2 : BOOL ;	//Anti-intrusion sensor 2 temp. reset memory/Mem.passage 0 ctl anti-intrusion 2
  xCMUT : BOOL ;	//Auxiliary bit of the CMUT rising edge/Bit aux. du front montant de CMUT
END_VAR
VAR_TEMP
  REMUT : BOOL ;	//Rising Edge of CMUT / Front Montant de CMUT
END_VAR
BEGIN
// body was compiled from another editor; compiled code not shown
END_FUNCTION_BLOCK

FUNCTION_BLOCK "BFS_BIMA1"	// FB 1721
//**********************************************************************
//*                             BFS_BIMA1                              *
//**********************************************************************
//(in english further below)
//DESCRIPTION: 
//************ 
//Le FB1721 "BFS_BIMA1" est un relais de securite logiciel programme en Step7 + 
//Distributed Safety pour assurer la surete de fonctionnement d'une bi-manuelle 
//geree par automate Simatic Failsafe.
//
//Son role est 
//"De piloter une information de validation de la bi-manuelle utilisee par le 
//programme de securite pour gerer des energies de commande ou/et de puissance 
//securisees 
//"De controler l'appui simultane sur les deux boutons
//"De controler a chaque cycle la retombee des deux boutons 
//
//C'est une evolution du FB1721 "BFS_BIMA1".
//
//Pas de bloc associe pour le diagnostic via IHMP+
//
//*************************English Information*******************************
//Description
//***********
//The FB1719 "BFS_BIMA" is a software safety relay in Step 7 + Distributed 
//Safety to ensure the dependability of a two-hands control managed by a Simatic 
//Failsafe PLC.
//
//It serves: 
//"to control an information of validation of the two-hand control used by the 
//safety program in order to manage the safe energies of control or/and power.
//"to check the concurrently pressing of both buttons
//"to check at each cycle the releasing of both buttons
//
//It's an evolution of FB1721 "BFS_BIMA1".
//
//No associated block for the diagnostics via IHMP+
//
AUTHOR : RENAULT
FAMILY : RENAULT
NAME : BIMA1
VERSION : 1.0
VAR_INPUT
  AT : BOOL ;	//Operator Work Authorization/Autorisation Travail operateur
  ET : BOOL ;	//Operator Completion/Enregistrement Travail Operateur
  BVOp11_NO : BOOL ;	//Pushbutton 1 Channel 1 NO contact/BP1 Voie 1 contact NO
  BVOp12_NC : BOOL ;	//Pushbutton 1 Channel 2 NC contact/BP1 Voie 2 contact NC
  BVOp21_NO : BOOL ;	//Pushbutton 2 Channel 1 NO contact/BP2 Voie 1 contact NO
  BVOp22_NC : BOOL ;	//Pushbutton 2 Channel 1 NC contact/BP2 Voie 2 contact NC
END_VAR
VAR_OUTPUT
  MRBVOp : BOOL ;	//Memory of the validation pushbuttons releasing/Mem. retombee BP de validatio
  Q : BOOL ;	//Two hand control validation/Validation bi-manuelle
END_VAR
VAR
  x : BOOL ;	//Bit of instance location/Bit de localisation de l'instance
  TON : FB 185;	//Simultaneity timer/Tempo de controle de la simultaneite
  MRBVOp_TIA : BOOL ;	//Memory of the validation pushbuttons releasing/Mem. retombee BP de validatio
  Q_TIA : BOOL ;	//Two hand control validation/Validation bi-manuelle
END_VAR
VAR_TEMP
  B0 : BOOL ;	//Released pushbuttons/Boutons poussoirs relaches
  B1 : BOOL ;	//Activated first pushbutton/Bouton poussoir 1 active
  B2 : BOOL ;	//Activated second pushbutton/Bouton poussoir 2 active
END_VAR
BEGIN
// body was compiled from another editor; compiled code not shown
END_FUNCTION_BLOCK

// FC 1100: know-how protected block, not included

FUNCTION "0_00_TSCYCLE" : VOID	// FC 1101
VERSION : 0.1
BEGIN
// body was compiled from another editor; compiled code not shown
END_FUNCTION

// DB 1100: know-how protected block, not included

// DB 1110: know-how protected block, not included

// DB 1111: know-how protected block, not included

// DB 1112: know-how protected block, not included

// DB 1113: know-how protected block, not included

DATA_BLOCK "TSM"	// DB 1279
VERSION : 0.1
  STRUCT
   Z1_S_QBAD : BOOL ;	//Z1: SAFETY MODULE FAULT / DEFAUT MODULE DE SECURITE
   Z1_CRM_DEF : BOOL ;	//Z1: FAULT EARTH CONNEXION CONTROL / DEFAUT RELAI CONTROLE MISE A LA MASSE ALIM
   Z1_IBFF : BOOL ;	//Z1: SAFETY CIRCUIT CORRECT WORKING INFO / INFO BON FONCTIONNEMENT FILERIE
   Z1AU_SECU : BOOL ;	//Z1: EMERGENCY STOP ELECTRICAL COMMON / COMMUN ELECTRIQUE ARRET D URGENCE
   Z1AU_SECU_OK : BOOL ;	//Z1: EMERGENCY STOP ELECTRICAL COMMON OK / COMMUN ELECTRIQUE ARRET D URGENCE OK
   Z1_AU_DEF : BOOL ;	//Z1: FAULT EMERGENCY STOP COMMON (AU) / DEFAUT COMMUN ARRET D URGENCE (AU)
   Z1ES_SECU : BOOL ;	//Z1: START UP ELECTRICAL COMMON / COMMUN ELECTRIQUE MISE EN SERVICE
   Z1ES_SECU_OK : BOOL ;	//Z1: START UP ELECTRICAL COMMON OK / COMMUN ELECTRIQUE MISE EN SERVICE OK
   Z1_ES_DEF : BOOL ;	//Z1: FAULT START UP COMMON (ES) / DEFAUT COMMUN MISE EN SERVICE (ES)
   Z1FZ_SECU : BOOL ;	//Z1: ZONE CLOSED ELECTRICAL COMMON / COMMUN ELECTRIQUE FEMETURE ZONE
   Z1FZ_SECU_OK : BOOL ;	//Z1: ZONE CLOSED ELECTRICAL COMMON OK / COMMUN ELECTRIQUE FEMETURE ZONE OK
   Z1_FZ_DEF : BOOL ;	//Z1: FAULT CLOSED ZONE COMMON (FZ)/DEFAUT COMMUN FERMETURE ZONE (FZ)
   Z1AIR_SECU : BOOL ;	//Z1: AIR ELECTRICAL COMMON / COMMUN ELECTRIQUE AIR
   Z1AIR_SECU_OK : BOOL ;	//Z1: AIR ELECTRICAL COMMON OK / COMMUN ELECTRIQUE AIR OK
   Z1_AIR_DEF : BOOL ;	//Z1: FAULT AIR PRESSURE (7 BAR) / DEFAUT PRESSION D AIR (7 BAR)
   Z1FZTR_SECU : BOOL ;	//Z1: TEMPO ZONE CLOSED ELECTRICAL COMMON / COMMUN ELEC FEMETURE ZONE TEMPORISE
   Z1FZTR_SECU_OK : BOOL ;	//Z1: TEMPO ZONE CLOSED ELECTRICAL COMMON OK / COMMUN ELEC FEMETURE ZONE OK TEMPO
   Z1_FZTR_DEF : BOOL ;	//Z1: FAULT CLOSED ZONE TEMPORISED COMMON/DEF COMMUN FERMETURE ZONE TEMPORISE
   ECH_AUOK_AMONT : BOOL ;	//FACILITY: EXCHANGE WITH UPSTREAM FACILITY - EMERGENCY STOP OK / AU OK->ILOT AM
   ECH_ESOK_AMONT : BOOL ;	//FACILITY: EXCHANGE WITH UPSTREAM FACILITY - POWER ON OK / ES OK->ILOT AM
   ECH_FZOK_AMONT : BOOL ;	//FACILITY: EXCHANGE WITH UPSTREAM FACILITY - CLOSED ZONE OK / FZ OK->ILOT AM
   SEND_ERROR_AMONT : BOOL ;	//FACILITY: EXCHANGE WITH UPSTREAM FACILITY- SEND ERROR/ ERREUR EMIS-> ILOT AM
   SEND_SUBS_ON_AMONT : BOOL ;	//FACILITY: EXCHANGE UPSTREAM FACILITY- EMISSION SUBSTITUTION/ SUBS EMIS->ILOT AM
   RECV_ACK_REI_AMONT : BOOL ;	//FACILITY: EXCHANGE WITH UPSTREAM FACILITY- RECEPTION ACK/ ACQ RECEPTION->ILO AM
   RECV_ERROR_AMONT : BOOL ;	//FACILITY: EXCHANGE WITH UPSTREAM FACILITY- RECV ERROR/ ERREUR RECEPT-> ILOT AM
   RECV_SUBS_ON_AMONT : BOOL ;	//FACILITY: EXCHANGE UPSTREAM FACILITY- RECEPT SUBSTITUTION/ SUBS RECEPT->ILOT AM
   RECV_ACK_REQ_AMONT : BOOL ;	//FACILITY: EXCHANGE UPSTREAM FACILITY- RECEPT REQ ACK/ ACQ REQ RECEPTION->ILO AM
   RECV_SENDMODE_AMONT : BOOL ;	//FACILITY: SEND/RECV MODE WITH UPSTREAM FACILITY / MODE EMIS/RECEPT->ILOT AM
   ECH_AUOK_AVAL : BOOL ;	//FACILITY: EXCHANGE WITH DOWNSTREAM FACILITY- EMERGENCY STOP OK / AU OK->ILOT AV
   ECH_ESOK_AVAL : BOOL ;	//FACILITY: EXCHANGE WITH DOWNSTREAM FACILITY - POWER ON OK / ES OK->ILOT AV
   ECH_FZOK_AVAL : BOOL ;	//FACILITY: EXCHANGE WITH DOWNSTREAM FACILITY - CLOSED ZONE OK / FZ OK->ILOT AV
   SEND_ERROR_AVAL : BOOL ;	//FACILITY: EXCHANGE WITH DOWNSTREAM FACILITY- SEND ERROR/ ERREUR EMIS-> ILOT AV
   SEND_SUBS_ON_AVAL : BOOL ;	//FACILITY: EXCHANGE DOWNSTREAM FACILITY- EMISSION SUBS/ SUBS EMIS->ILOT AV
   RECV_ACK_REI_AVAL : BOOL ;	//FACILITY: EXCHANGE WITH DOWNSTREAM FACILITY- RECEPT ACK/ ACQ RECEPTION->ILOT AV
   RECV_ERROR_AVAL : BOOL ;	//FACILITY: EXCHANGE WITH DOWNSTREAM FACILITY- RECV ERROR/ ERREUR RECEPT->ILOT AV
   RECV_SUBS_ON_AVAL : BOOL ;	//FACILITY: EXCHANGE DOWNSTREAM FACILITY- RECEPT SUBS/ SUBS RECEPT->ILOT AV
   RECV_ACK_REQ_AVAL : BOOL ;	//FACILITY: EXCHANGE DOWNSTREAM FACILITY- RECEPT REQ ACK/ ACQ REQ RECEP->ILOT AV
   RECV_SENDMODE_AVAL : BOOL ;	//FACILITY: SEND/RECV MODE WITH DOWNSTREAM FACILITY / MODE EMIS/RECEPT->ILOT AV
   B0_Secu_OK : BOOL ;	//Z1: B0 Contacteur chaine Sécurité OK
   B0CR_Def : BOOL ;	//Z1: Def. Retour contacteur chaine meuble B0
   B1CR_Def : BOOL ;	//Z1: Def. Retour contacteur chaine meuble B1
   G0SOP_Secu : BOOL ;	//G0:  Commande Boucle Sécurité Opérateur
   G0SOP_Secu_OK : BOOL ;	//G0:  Boucle Sécurité Opérateur OK
   G0SOP_Def : BOOL ;	//G0: Def. SOP
   P0SOP_Secu : BOOL ;	//P0:  Commande Boucle Sécurité Opérateur
   P0SOP_Secu_OK : BOOL ;	//P0:  Boucle Sécurité Opérateur OK
   P0SOP_Def : BOOL ;	//P0: Defaut Boucle Sécurité Opérateur
   P01SOP_Secu : BOOL ;	//P01: Commande Boucle Sécurité Opérateur
   P01SOP_Secu_OK : BOOL ;	//P01:  Boucle Sécurité Opérateur OK
   P01SOP_Def : BOOL ;	//P01: Def. SOP
   P02SOP_Secu : BOOL ;	//P02: Commande Boucle Sécurité Opérateur
   P02SOP_secu_OK : BOOL ;	//P02:  Boucle Sécurité Opérateur OK
   P02SOP_Def : BOOL ;	//P02: Def. SOP
   P1SOP_Secu : BOOL ;	//P1:  Commande Boucle Sécurité Opérateur
   P1SOP_Secu_OK : BOOL ;	//P1:  Boucle Sécurité Opérateur OK
   L1RLV_Secu : BOOL ;	//Z1: Commande Relais De Ligne variateur L1
   L1RLV_Secu_OK : BOOL ;	//Z1: Relais De Ligne variateur L1
   L1RLV_Def : BOOL ;	//Z1: Def. Relais De Ligne variateur L1
   L1RL_Secu_OK : BOOL ;	//Z1: Relais De Ligne élévateur L1
   L1RL_Def : BOOL ;	//Z1: Def. Relais De Ligne élévateur L1
   L2RLV_Secu : BOOL ;	//Z1: Commande Relais De Ligne Translateur L2 OK
   L2RLV_Secu_OK : BOOL ;	//Z1: Relais De Ligne Translateur L2 OK
   L2RLV_Def : BOOL ;	//Z1: Def. Relais De Ligne Translateur L2
   L3RLV_Secu : BOOL ;	//Z1: Commande Relais De Ligne élévateur L3
   L3RLV_Secu_OK : BOOL ;	//Z1: Relais De Ligne élévateur L3 OK
   L3RLV_Def : BOOL ;	//Z1: Def. Relais De Ligne élévateur L3
   L3RL_Secu_OK : BOOL ;	//Z1: Relais De Ligne élévateur L3 OK
   L3RL_Def : BOOL ;	//Z1: Def. Relais De Ligne élévateur L3
   P0Pos_Def : BOOL ;	//P0: Def. Position Plateau
   V0RLV_Secu : BOOL ;	//Z1: Commande Relais De Ligne élévateur V0
   V0RLV_Secu_OK : BOOL ;	//Z1: Relais De Ligne élévateur V0 OK
   V0RLV_Def : BOOL ;	//Z1: Def. Relais De Ligne élévateur V0
   V0RLVVE_OK : BOOL ;	//Z1: Relais De Ligne verrou élévateur V0
   V0RLVVE_Def : BOOL ;	//Z1: Def. Relais De Ligne verrou élévateur V0
   F1MRBV : BOOL ;	//F1_Ope: Mémoire Retombée Boutons Validations
   F2MRBV : BOOL ;	//F2_Ope: Mémoire Retombée Boutons Validations
   F3MRBV : BOOL ;	//F3_Ope: Mémoire Retombée Boutons Validations
   F1BIM_Q : BOOL ;	//F1_Ope: Sortie Bimanuelle
   F2BIM_Q : BOOL ;	//F2_Ope: Sortie Bimanuelle
   F3BIM_Q : BOOL ;	//F3_Ope: Sortie Bimanuelle
   C0SOP_Secu : BOOL ;	//C0: Commande Boucle Sécurité Opérateur
   C0SOP_Secu_OK : BOOL ;	//C0: Boucle Sécurité Opérateur OK
   C0SOP_Def : BOOL ;	//C0: Défaut Boucle Sécurité Opérateur
   F0SOP_Secu : BOOL ;	//F0: Commande Boucle Sécurité Opérateur
   F0SOP_Secu_OK : BOOL ;	//F0: Boucle Sécurité Opérateur OK
   F0SOP_Def : BOOL ;	//F0: Défaut Sécurité Opérateur F0
   R1SOPR_Secu : BOOL ;	//R1: Commande Boucle Sécurité Opérateur Robot
   R1SOPR_Secu_OK : BOOL ;	//R1: Boucle Sécurité Opérateur Robot OK
   R1SOPR_Def : BOOL ;	//R1: Défaut Sécurité Opérateur Robot
  END_STRUCT ;	
BEGIN
END_DATA_BLOCK

// DB 1286: know-how protected block, not included

// DB 1287: know-how protected block, not included

// DB 1288: know-how protected block, not included

// DB 1289: know-how protected block, not included

// DB 1300: know-how protected block, not included

SYMBOL_TABLE
"I01"	DB 1	FB 1	// FACILITY: INSTANCE DB (FB1)
"I02"	DB 2	FB 2	// FACILITY: INSTANCE DB FOR MMC CONTROL (FB2)
"I03"	DB 3	FB 3	// FACILITY: INSTANCE DB FOR MOP/LOP
"I04"	DB 4	FB 4	// FACILITY: INSTANCE DB FOR COMMUNICATION / DB D'INSTANCE POUR LA COMMUNICATION
"SFM_DB"	DB 75	FB 20	// FACILITY: DB FAILURE MESSAGE (SFM_FB) LINK WITH PROFINET CONTROL
"SFM_GLOBAL_DB"	DB 76	DB 76	// DIAGNOSTIC BLOCK FOR THE SIGNALISATION OF THE SYSTEM ERRORS
"SFM_PN"	DB 77	DB 77	// PROFINET DIAGNOSTIC FUNCTION EDITING DB FOR IHMP
"SIP1"	DB 89	DB 89	// SIPTOL EXCHANGES DATAS / TABLE D'ECHANGES SIPTOL
"PILE"	DB 90	DB 90	// FACILITY: FIFO STORAGE / PILE DE STOCKAGE
"CAB"	DB 91	DB 91	// L0: BARCODE READER DB / DB LECTEUR CODE BARRE
"IDENT"	DB 93	DB 93	// RFID DATAS / IDENTIFIANT DYNAMIQUE
"POS"	DB 94	DB 94	// Posiciones de giro
"IIT"	DB 96	DB 96	// FACILITY: PART TABLE / DB TABLE PIECE
"IIS"	DB 97	DB 97	// FACILITY: SUPPORT WORD TABLE / DB MOTS SUPPORT
"IG"	DB 99	DB 99	// FACILITY: GLOBAL DB / DB GLOBAL
"Z1"	DB 100	FB 100	// ZONE 1: INSTANCE DB
"Z1A0"	DB 101	FB 101	// A0 MONTAGE INSTANCE DATA BLOC / BLOC DE DONNEES INSTANCE A0 MONTAGE
"Z1A1"	DB 104	FB 104	// A1 OP_BPVAL INSTANCE DATA BLOC / BLOC DE DONNEES INSTANCE A1 OP_BPVAL
"Z1A2"	DB 105	FB 105	// A2 OP_BPVAL INSTANCE DATA BLOC / BLOC DE DONNEES INSTANCE A2 OP_BPVAL
"AUX_SEW"	DB 111	DB 111
"Z1T"	DB 198	DB 198	// ZONE 1: REFERENCE TIME FOR MOVEMENTS
"Z1G"	DB 199	DB 199	// ZONE 1: GLOBAL DB
"Z2"	DB 200	FB 200	// ZONE 1: INSTANCE DB
"Z2B0"	DB 210	FB 210	// B0 MONTAGE INSTANCE DATA BLOC / BLOC DE DONNEES INSTANCE B0 MONTAGE
"Z2B1"	DB 211	FB 211	// B1 OP_BPVAL INSTANCE DATA BLOC / BLOC DE DONNEES INSTANCE B1 OP_BPVAL
"Z2B2"	DB 212	FB 212	// B2 OP_BPVAL INSTANCE DATA BLOC / BLOC DE DONNEES INSTANCE B2 OP_BPVAL
"Z2T"	DB 298	DB 298	// ZONE 2: REFERENCE TIME FOR MOVEMENTS
"Z2G"	DB 299	DB 299	// ZONE 2: GLOBAL DB
"ITS0"	DB 1100	FB 1100	// ILOT : DB INSTANCE FB1100
"ITSZ1_AU_ES_FZ"	DB 1110	FB 1110	// Z1 : DB D'INSTANCE DU FB 1110
"ITSZ1SOP"	DB 1111	FB 1111	// Zone 1 : Operator safety
"ITSZ1VAR"	DB 1113	FB 1113	// Z1 : DB D'INSTANCE DU FB 1113
"ITSZ2_AU_ES_FZ"	DB 1120	FB 1120	// Zone 2 : common control
"ITSZ2SOP"	DB 1121	FB 1121	// Zone 2 : Operator safety
"ITSZ3_AU_ES_FZ"	DB 1130	FB 1130	// Zone 3 : common control
"ITSZ3SOP"	DB 1131	FB 1131	// Zone 3 : Operator safety
"ITSZ2_AU_ES_FZ."	DB 1210	FB 1210	// Z2 : DB D'INSTANCE DU FB 1210
"ITSZ2SOP."	DB 1211	FB 1211	// Zone 2 : Operator safety
"TSM"	DB 1279	DB 1279
"TSE_AMONT"	DB 1286	FB 1692	// STD - INSTANCE DB OF FB 1692 (F_SENDDP) SAFETY DATA SEND
"TSR_AMONT"	DB 1287	FB 1693	// STD - INSTANCE DB OF FB 1693 (F_RCVDP) SAFETY DATA RECEIVE
"TSE_AVAL"	DB 1288	FB 1692	// STD - INSTANCE DB OF FB 1692 (F_SENDDP) SAFETY DATA SEND
"TSR_AVAL"	DB 1289	FB 1693	// STD - INSTANCE DB OF FB 1693 (F_RCVDP) SAFETY DATA RECEIVE
"F_GLOBDB"	DB 1300	DB 1300	// F_: F_Global_Data Block
"F00030__Z1ZB_M13"	DB 1301	FB 1300
"F00036__Z1ZB_M14"	DB 1302	FB 1300
"F00312_PROFIsafe_telegra"	DB 1303	FB 1300
"F00068_FVDO_P2__3DO_F"	DB 1304	FB 1300
"F00353_PROFIsafe_16_E_S"	DB 1305	FB 1300
"F00013__Z1ZB_M11"	DB 1307	FB 1300
"F00019__Z1ZB_M12"	DB 1308	FB 1300
"F00025__Z1ZB_M15"	DB 1309	FB 1300
"F00417__Z2ZB_M12"	DB 1319	FB 1300
"F00423__Z2ZB_M13"	DB 1320	FB 1300
"F00411__Z2ZB_M11"	DB 1321	FB 1300
"F00405__Z2ZB_M10"	DB 1322	FB 1300
"F00294__Z1SPA2"	DB 1325	FB 1300
"F01170__C02S1"	DB 1327	FB 1300
"F00305__Z2SPA1"	DB 1328	FB 1300
"F00316__Z2SPA2"	DB 1329	FB 1300
"F01010__B02S1"	DB 1330	FB 1300
"F00979__B01S1"	DB 1331	FB 1300
"F00327__Z3SPA1"	DB 1332	FB 1300
"F00338__Z3SPA2"	DB 1333	FB 1300
"F01138__C01S1"	DB 1334	FB 1300
"F01202__C03S1"	DB 1336	FB 1300
"F01514_A1LAS"	DB 1337	FB 1300
"F01524_B1LAS"	DB 1338	FB 1300
"F01534_C1LAS"	DB 1339	FB 1300
"F00618__B2IM_M03"	DB 1351	FB 1300
"AFF"	DB 1863	DB 1863	// SIEBERT DISPLAY STRING STORAGE / STOCKAGE MESSAGE AFFICHEUR SIEBERT
"DB_IHM_WINCC"	DB 1962	FB 1962	// FACILITY: HMI INTERFACING WINCCFLEXIBLE RT
"DB_MMC"	DB 2000	DB 2000	// BACKUP COPY AND RESTORE OF EXTERN MEMORY MAP (MMC)
"DB_PN"	DB 2036	FB 2036	// INSTANCE IO PROFINET DB
"0_01_ILOT"	FB 1	FB 1	// FACILITY: FACILITY MANAGEMENT
"0_02_MMC"	FB 2	FB 2	// FACILITY: BACKUP MANAGEMENT AND DATA RESTITUTION ON EXTERNAL MMC CARD
"0_03_XOP"	FB 3	FB 3	// FACILITY: MOP/LOP MANAGEMENT
"0_04_COM"	FB 4	FB 4	// FACILITY: COM CONTROL WITH SIPTOL / GESTION DE LA COMMUNICATION AVEC SIPTOL
"SFM_FB"	FB 20	FB 20	// DIAGNOSTIC BLOCK FOR SYSTEM ERRORS SIGNALLING
"1_00_ZONE1"	FB 100	FB 100	// ZONE 1: ZONE CONTROL
"1_A0_MONTAGE"	FB 101	FB 101	// A0 MONTAGE FUNCTION BLOC / SECTION PROGRAMME A0 MONTAGE
"1_A1_OP_BPVAL"	FB 104	FB 104	// A1 OP_BPVAL FUNCTION BLOC / SECTION PROGRAMME A1 OP_BPVAL
"1_A2_OP_BPVAL"	FB 105	FB 105	// A2 OP_BPVAL FUNCTION BLOC / SECTION PROGRAMME A2 OP_BPVAL
"F_TON"	FB 185	FB 185	// F_: Timer Switch On Delay
"F_TOF"	FB 186	FB 186	// F_: Timer Switch Off Delay
"F_2HAND"	FB 188	FB 188	// F_: Two Hand Monitoring
"F_1oo2DI"	FB 190	FB 190	// F_: 1oo2 Evaluation with Discrepancy Analysis
"2_00_ZONE2"	FB 200	FB 200	// ZONE 2: ZONE CONTROL
"2_B0_MONTAGE"	FB 210	FB 210	// B0 MONTAGE FUNCTION BLOC / SECTION PROGRAMME B0 MONTAGE
"2_B1_OP_BPVAL"	FB 211	FB 211	// B1 OP_BPVAL FUNCTION BLOC / SECTION PROGRAMME B1 OP_BPVAL
"2_B2_OP_BPVAL"	FB 212	FB 212	// B2 OP_BPVAL FUNCTION BLOC / SECTION PROGRAMME B2 OP_BPVAL
"TS0"	FB 1100	FB 1100	// ILOT: FB Gestion SAFETY ilot
"TSZ1_AU_ES_FZ"	FB 1110	FB 1110
"TSZ1_SOP"	FB 1111	FB 1111	// ZONE 1 : FB Gestion SAFETY  SOP de la zone 1
"TSZ1_VAR"	FB 1113	FB 1113
"TSZ2_AU_ES_FZ"	FB 1210	FB 1210
"TSZ2_SOP"	FB 1211	FB 1211	// ZONE 2 : FB Gestion SAFETY  SOP de la zone 2
"F_IO_CGP"	FB 1300	FB 1300	// F_: Driver Block In-Output with Channel Granular Passivation
"F_CTRL_1"	FB 1301	FB 1301	// F_: Test Block an Programm Run Control 1
"F_CTRL_2"	FB 1302	FB 1302	// F_: Test Block an Programm Run Control 2
"FITON"	FB 1303	FB 1303
"FIACK_GL"	FB 1304	FB 1304
"FI1oo2DI"	FB 1305	FB 1305	// FI: 1oo2 Evaluation with Discrepancy Analysis
"F_DIAG_N"	FB 1307	FB 1307	// F_: Diagnosticbuffer Message with non CPU-Stop
"F_RTGCO2"	FB 1308	FB 1308
"BF_DEVERM"	FB 1649	FB 1649	// BF STAGE DRY RUN CONTROL / BF GESTION DEVERMINAGE POSTE
"BF_RB_NISSAN"	FB 1650	FB 1650	// FANUC NISSAN ROBOT FB / BF ROBOT FANUC NISSAN
"TUSEND"	FB 1681	FB 1681	// Send Data via UDP
"TCON"	FB 1685	FB 1685	// Connect
"F_SENDDP"	FB 1692	FB 1692	// F_: Send Data via PROFIBUS DP / PROFINET IO
"F_RCVDP"	FB 1693	FB 1693	// F_: Receive Data via PROFIBUS DP / PROFINET IO
"F_ACK_GL"	FB 1695	FB 1695	// Acquittement global de toutes les périphéries F d'un groupe d'exécution F
"P_SEND"	FB 1698	FB 1698	// Send Data to CP340
"P_RCV"	FB 1699	FB 1699	// Receive Data from CP340
"BFS_BSEC1"	FB 1710	FB 1710
"BFS_BSECTR1"	FB 1711	FB 1711
"BFS_PORTE1"	FB 1712	FB 1712
"BFS_AIR1"	FB 1713	FB 1713
"BFS_CRM1"	FB 1714	FB 1714
"BFS_CR1"	FB 1715	FB 1715
"BFS_CAME_ROBOT1"	FB 1716	FB 1716
"BFS_MUT1"	FB 1717	FB 1717
"BFS_ROB_KUKA_PS"	FB 1720	FB 1720
"BFS_BIMA1"	FB 1721	FB 1721
"BF_NC_LOCATOR_16-32"	FB 1827	FB 1827	// GESTION DES NC_LOCATOR
"BF_MULTIPOS"	FB 1833	FB 1833	// COMMANDE MOUVEMENT MANUT HORIZONTAL ET VERTICALE JUSQU'A 16 POSITIONS
"BF_PNPN_MESG"	FB 1852	FB 1852	// SEND RECEIVE MESSAGE BY PNPN INTERFACE/ EMISSION RECEPTION MESSAGE VIA PNPN
"BF_G120DS_V2"	FB 1853	FB 1853	// G120D DRIVE BOX CONTROL / GESTION COFFRET VAR G120D
"BF_G120S_V2"	FB 1854	FB 1854	// G120 DRIVE PLATE CONTROL / GESTION PLATINE VAR G120
"BF_CARACT_SIEBERT"	FB 1856	FB 1856	// SIEBERT DISPLAY MESSAGE CONFIGURATION / MISE EN FORME MESSAGE AFFICHEUR SIEBERT
"BF_RECALAGE2"	FB 1857	FB 1857	// BF ASSOCIEE AU POINT DE GESTION DE FLUX "RECALAGE"
"BF_LANCEMENT"	FB 1858	FB 1858	// GESTION LANCEMENT SIPTOL
"BF_AFF SIEBERT (2*13) PN"	FB 1860	FB 1860	// AFFICHEUR 2 LIGNES DE 13 CARACTERES
"BF_WELDING_BOX"	FB 1868	FB 1868	// WELDING BOX CONTROL / GESTION DES COFFRETS PARAMETRES SOUDURE
"BF_CONF_MACHINE"	FB 1869	FB 1869	// GESTION BASE DE DONNEE CONFIGURATION MACHINE
"BF_CODE_PROCESS"	FB 1870	FB 1870	// GESTION BASE DE DONNEE CODE PROCESS
"BF_DATABASE3"	FB 1871	FB 1871	// DATABASE MANAGEMENT / GESTION BASE DE DONNEES
"BF_IHMMUT1"	FB 1874	FB 1874	// Diagnostic IHM(P) BFS_MUT1
"BF_IHMCAME_ROBOT1"	FB 1875	FB 1875	// BF gérant le bon fonctionnement de la came robot
"BF_IHMCR1"	FB 1876	FB 1876	// BF gérant l'IHM du relais non piloté par l'API mais controlé
"BF_IHMCRM1"	FB 1877	FB 1877	// BF gérant l'IHM du relais de controçle raccordement de masse CRM
"BF_S120_S"	FB 1892	FB 1892	// Commande d'un axe S120 en mode Positionnement
"BF_CABRS"	FB 1897	FB 1897	// BARCODE READER / LECTEUR DE CODE A BARRE
"BF_IHMPORTE1"	FB 1930	FB 1930	// BF - ZONE : Diagnostic du bloc BFS_IHMPORTE
"BF_IHMAIR1"	FB 1931	FB 1931	// BF - ZONE : Diagnostic du bloc BFS_IHMAIR
"BF_ZONE_MODE_IHM1"	FB 1932	FB 1932	// Zone: Traitement des Modes et des pupitre de cde manu de la  zone
"BF_RB_COD_PREH_API"	FB 1953	FB 1953	// Gestion du préhenseur par API (séquences 1 à 16)
"BF_MODBUS_MASTER_CP340"	FB 1958	FB 1958	// MODBUS MAITRE SUR CP 340 (LIAISON SERIE)
"BF_MODBUS_SLAVE_CP340"	FB 1959	FB 1959	// MODBUS ESCLAVE AVEC CP340
"BF_MODBUS_TCPIP_MASTER"	FB 1960	FB 1960	// BF gerant le protocole MODBUS TCP/IP en tant que Client TCP et Maitre MODBUS
"BF_MODBUS_TCPIP_SLAVE"	FB 1961	FB 1961	// ESCLAVE MODBUS SUR CP ETHERNET
"BF_IHM_WINCC"	FB 1962	FB 1962	// BF- GESTION IMAGES WINCC FLEXIBLE
"BF_RB_SERVICE"	FB 1997	FB 1997	// BF- Envoi d'un groupe de robot en rodage
"BF_MMC"	FB 2000	FB 2000	// SAUVEGARDE ET RESTITUTION MEMOIRE SUR CARTE MEMOIRE EXTERNE (MMC)
"BF_MB_CHAINE1"	FB 2001	FB 2001	// PILOTAGE DU MOTEUR DU MEUBLE ET SURVEILLANCE DES DEFAUTS
"BF_MB_BUTEE1"	FB 2002	FB 2002	// MEUBLE A ACCUMULATION - PILOTAGE D'UNE BUTEE
"BF_MARIAGE_API"	FB 2003	FB 2003	// Gestion des Mariages Pièces
"BF_ILOT"	FB 2004	FB 2004	// BF- GESTION INFO LIE A L'INSTALLATION (ILOT)
"BF_B_VIEAPI"	FB 2006	FB 2006	// CONTRÔLE DE LA COMMUNICATION ENTRE DEUX AUTOMATES EN LIAISON
"BF_BUTEE_CONVOYEUR2"	FB 2007	FB 2007	// PILOTAGE D'UNE BUTEE
"BF_IDENT"	FB 2015	FB 2015	// LECTURE/ECRITURE DES ETIQUETTES RFID
"BF_ROBOT"	FB 2016	FB 2016	// Interface API - Robot Version 1.2a
"BF_TCY_SUIV"	FB 2019	FB 2019	// MESURE LES TEMPS DE CYCLE D'UN MOYEN DE PRODUCTION
"BF_RUP_FLU"	FB 2020	FB 2020	// SUIVI-RUPTURE DE FLUX
"BF_CPT_PIECE"	FB 2021	FB 2021	// BF- COMPTEUR DE PIECE
"BF_API_MAITRE_CAL"	FB 2031	FB 2031	// Gestion du Dialogue API MAITRE CAL
"BF_ACT_DESACT"	FB 2033	FB 2033	// BF- ACTIVATION DESACTIVATION D'UN IO DEVICE
"BF_DIAG_PROFINET"	FB 2036	FB 2036	// BF- DIAGNOSTIC PROFINET IO
"BF_TF_TP"	FB 2037	FB 2037	// TRANSFERT DE TABLE DE MEMOIRES PIECES
"BF_FIFO"	FB 2039	FB 2039	// ASSURE LA GESTION D'UNE PILE FIFO
"BF_MVSE2P1"	FB 2040	FB 2040	// GESTION D'UN MOUVEMENT SIMPLE EFFET 2 POSITIONS
"BF_MOUVMP1"	FB 2041	FB 2041	// GESTION D'UN MOUVEMENT MULTI POSITION
"BF_MOUV2P1"	FB 2042	FB 2042	// BF- GESTION D'UN MOUVEMENT A 2 POSITIONS
"0_00_CYCLE_ILOT"	FC 1	FC 1	// FACILITY: CALL OF FACILITY FB
"fb185"	FC 2	FC 2
"SFM_FC"	FC 22	FC 22	// BLOCK DIAGNOSTIC FOR ERROR REPORTING SYSTEM
"1_00_CYCLE_Z1"	FC 100	FC 100	// ZONE 1: CALL OF FB ZONE
"2_00_CYCLE_Z2"	FC 200	FC 200	// ZONE 2: CALL OF FB ZONE
"3_00_CYCLE_Z3"	FC 300	FC 300	// ZONE 3: CALL OF FB ZONE
"0_00_TSSAFETY"	FC 1100	FC 1100	// STD - FACILITY: EXECUTION F GROUP ASSOCIATE TO OB32 (NORMAL TASK)
"0_00_TSCYCLE"	FC 1101	FC 1101	// CALL OPERATOR NOT IN ZONE FB LINKED IN FACILITY
"C_CNTRL"	FC 1697	FC 1697	// Read Connection Diagnostic Information
"AG_SEND"	FC 1698	FC 1698	// AG SEND
"AG_RECV"	FC 1699	FC 1699	// AG RECEIVE
"BADI"	I 0.0	BOOL	// (MOP-IM.M01-02): BOTON RESET FALLAS
"BRI"	I 0.1	BOOL	// (MOP-IM.M01-02): BOTON REARME DE ISLA
"BMCY"	I 0.2	BOOL	// (MOP-IM.M01-02): BOTON FUNCIONAMIENTO DE CICLO
"SMM"	I 0.3	BOOL	// (MOP-IM.M01-02): SELETOR MODE MANUAL
"SMA"	I 0.4	BOOL	// (MOP-IM.M01-02): SELETOR MODE AUTO
"Z1BMR1"	I 0.5	BOOL	// (MOP-IM.M01-02): BOTON RETROCESO MOVIMENTO
"Z1BMA1"	I 0.6	BOOL	// (MOP-IM.M01-02): BOTON AVANCE MOVIMENTO
"Z1CCAU"	I 10.0	BOOL	// (Z1ZB.M02): CONTROL RETORNO COMUN SEGURIDAD AU
"Z1CCES"	I 10.1	BOOL	// (Z1ZB.M02): CONTROL RETORNO COMUN SEGURIDAD ES
"Z1CCFZ"	I 10.2	BOOL	// (Z1ZB.M02): CONTROL RETORNO COMUN SEGURIDAD FZ
"Z1CCRL"	I 10.3	BOOL	// (Z1ZB.M02): CONTROL RETORNO COMUN SEGURIDAD RL
"Z1CCB24Z"	I 10.4	BOOL	// (Z1ZB.M02): RETORNO CONTROL DISJUNTOR 24V (24Z)
"Z1CCB24R"	I 10.5	BOOL	// (Z1ZB.M02): RETORNO CONTROL DISJUNTOR 24V (24R)
"Z1CCB24SC"	I 10.6	BOOL	// (Z1ZB.M02): RETORNO CONTROL DISJUNTOR 24V (SC)
"A0DPG1"	I 10.7	BOOL	// (Z1ZB.M02): Detector Presencia de Griper 1
"Z1CP7B"	I 11.0	BOOL	// (Z1ZB.M03): CONTROL PRESION 7 BARS
"Z1CRM"	I 11.1	BOOL	// (Z1ZB.M03): RETORNO RELE CONTROL DE MASA
"Z1CCB400_1"	I 11.2	BOOL	// (Z1ZB.M03): Breaker Control 400V (SDB1)
"Z1CRO_11"	I 11.3	BOOL	// (Z1ZB.M03): Safety Contactor Control 1 (SDB1)
"Z1CRO_12"	I 11.4	BOOL	// (Z1ZB.M03): Safety Contactor Control 2 (SDB1)
"Z1CCB400_2"	I 11.5	BOOL	// (Z1ZB.M03): Breaker Control 400V (SDB2)
"Z1CRO_21"	I 11.6	BOOL	// (Z1ZB.M03): Safety Contactor Control 1 (SDB2)
"Z1CRO_22"	I 11.7	BOOL	// (Z1ZB.M03): Safety Contactor Control 2 (SDB2)
"OP1VAL"	I 12.0	BOOL	// (Z1ZB.M04): Validacion OP1
"OP1BROC"	I 12.1	BOOL	// (Z1ZB.M04): Retorno Origen OP1
"A0DPG2"	I 12.3	BOOL	// (Z1ZB.M04): Detector Presencia de Griper 2
"OP2BROC"	I 12.6	BOOL	// (Z1ZB.M04): Retorno Origen OP2
"OP2VAL"	I 12.7	BOOL	// (Z1ZB.M04): Validacion OP2
"BAUI"	I 13.0	BOOL	// (Z1ZB.M11): PARADA DE ENERGENCIA ISLA
"BAU1"	I 13.1	BOOL	// (Z1ZB.M11): PARADA DE ENERGENCIA ZONA
"SSZ"	I 13.2	BOOL	// (Z1ZB.M11): SELETOR SEGURIDAD ZONA
"BAU2"	I 13.3	BOOL	// (Z1ZB.M11): PARADA DE ENERGENCIA ZONA
"A1SFF"	I 19.0	BOOL	// (Z1ZB.M12): Operator 1 SAFETY PEDAL EGS
"A2SFF"	I 19.1	BOOL	// (Z1ZB.M12): Operator 2 SAFETY PEDAL EGS
"EFC1"	I 19.2	BOOL	// (Z1ZB.M12): Presencia Estanteria EGS
"EFC2"	I 19.3	BOOL	// (Z1ZB.M12): Presencia Estanteria EGS
"A0BK1"	I 30.0	BOOL	// (Z1ZB.M013): Light Curtain 1 (For Trespassing )
"A0BK2"	I 30.1	BOOL	// (Z1ZB.M013): Light Curtain 2 (For Trespassing )
"A0BK3"	I 30.2	BOOL	// (Z1ZB.M013): Light Curtain 3 (For Trespassing )
"OP3CPOP1"	I 36.0	BOOL	// (Z1ZB.M014): Light Curtain 3 / laser 3 (CH1)
"OP3CPOP2"	I 36.1	BOOL	// (Z1ZB.M014): Light Curtain 3 / laser 3 (CH2)
"OP4CPOP1"	I 36.2	BOOL	// (Z1ZB.M014): Light Curtain 4 / laser 4 (CH1)
"OP4CPOP2"	I 36.3	BOOL	// (Z1ZB.M014): Light Curtain 4 / laser 4 (CH2)
"A2"	I 36.4	BOOL
"B2"	I 36.5	BOOL
"C2"	I 36.6	BOOL
"D2"	I 36.7	BOOL
"A0DRCH1"	I 60.0	BOOL	// DET MAG REC CH1
"A0DACH1"	I 60.1	BOOL	// DET MAG AV CH1
"A0DRSR51"	I 60.2	BOOL	// DET MAG REC SR51
"A0DASR51"	I 60.3	BOOL	// DET MAG AV SR51
"A0DAVR22"	I 60.4	BOOL	// DET MAG AV VR22
"A0DRVR22"	I 60.5	BOOL	// DET MAG REC VR22
"A0DRSR53"	I 60.6	BOOL	// DET MAG REC SR53
"A0DASR53"	I 60.7	BOOL	// DET MAG AV SR53
"A0DAVR32"	I 61.0	BOOL	// DET MAG AV VR32
"A0DRVR32"	I 61.1	BOOL	// DET MAG REC VR32
"A0DRSR4"	I 61.2	BOOL	// DET MAG REC SR4
"A0DASR4"	I 61.3	BOOL	// DET MAG AV SR4
"A0DAVR21"	I 61.4	BOOL	// DET MAG AV VR21
"A0DRVR21"	I 61.5	BOOL	// DET MAG REC VR21
"A0DRSR52"	I 61.6	BOOL	// DET MAG REC SR52
"A0DASR52"	I 61.7	BOOL	// DET MAG AV SR52
"A0DAVR31"	I 62.0	BOOL	// DET MAG AV VR31
"A0DRVR31"	I 62.1	BOOL	// DET MAG REC VR31
"A0DRSR54"	I 62.2	BOOL	// DET MAG REC SR54
"A0DASR54"	I 62.3	BOOL	// DET MAG AV SR54
"A0DRSR55"	I 62.4	BOOL	// DET MAG REC SR55
"A0DASR55"	I 62.5	BOOL	// DET MAG AV SR55
"A0DRSR61"	I 62.6	BOOL	// DET MAG REC SR61
"A0DASR61"	I 62.7	BOOL	// DET MAG AV SR61
"A0DRSR62"	I 63.0	BOOL	// DET MAG REC SR62
"A0DASR62"	I 63.1	BOOL	// DET MAG AV SR62
"A0DRSR63"	I 63.2	BOOL	// DET MAG REC SR63
"A0DASR63"	I 63.3	BOOL	// DET MAG AV SR63
"A0DRSR7"	I 63.4	BOOL	// DET MAG REC SR7
"A0DASR7"	I 63.5	BOOL	// DET MAG AV SR7
"A0DRSR65"	I 63.6	BOOL	// DET MAG REC SR65
"A0DASR65"	I 63.7	BOOL	// DET MAG AV SR65
"A0DRSR66"	I 64.0	BOOL	// DET MAG REC SR66
"A0DASR66"	I 64.1	BOOL	// DET MAG AV SR66
"A0DRSR91"	I 64.2	BOOL	// DET MAG REC SR91
"A0DASR91"	I 64.3	BOOL	// DET MAG AV SR91
"A0DRSR92"	I 64.4	BOOL	// DET MAG REC SR92
"A0DASR92"	I 64.5	BOOL	// DET MAG AV SR92
"A0DPP1"	I 66.0	BOOL	// DET PRESENCIA CANULA
"A0DPP2"	I 66.1	BOOL	// DET PRESENCIA PIEZA POT DETENTE
"A0DPP3"	I 66.2	BOOL	// DET PRESENCIA V3
"A0DPP4"	I 66.3	BOOL	// DET PRESENCIA PIEZA POT DETENTE
"A0DPP5"	I 66.4	BOOL	// DET PRESENCIA PIEZA POT DETENTE
"A0DPP6"	I 66.5	BOOL	// DET PRESENCIA TUBO V2-V3
"A0DPP7"	I 66.6	BOOL	// DET PRESENCIA TUBO V2-V3 B52
"A0DPP8"	I 66.7	BOOL	// DET PRESENCIA TUBO V2-V3 L52
"A0DPP9"	I 67.0	BOOL	// DET PRESENCIA PIEZA V2 TUBO K4M
"A0DPP10"	I 67.1	BOOL	// DET PRESENCIA PIEZA V2 TUBO K7Mk
"A0DPP11"	I 67.2	BOOL	// DET PRESENCIA DESCENSO TUBO
"A0DPP12"	I 67.3	BOOL	// DET PRESENCIA DESCENSO TUBO K7Mk
"A0DPP13"	I 67.4	BOOL	// DET PRESENCIA DESCENSO TUBO K4M
"A0DP6BAR"	I 67.6	BOOL	// DET PRESENCIA 6 BAR
"A0CCSOP"	I 68.0	BOOL	// (A0IM1-FVD0): Contro Comun SOP
"A0_CDJTR"	I 258.0	BOOL	// (A0SBS120): CONTROLE DISJONCTEUR 400V
"A0_CRFR"	I 258.1	BOOL	// (A0SBS120):CTRL RELAIS DE FREIN
"A0_CTRFR"	I 258.2	BOOL	// (A0SBS120):CTRL TEMPERATURE RESISTANCE DE FREINAGE
"A0_DI4"	I 258.3	BOOL	// (A0SBS120): DIGITAL INPUT 4
"A0_FCORR"	I 259.0	BOOL	// (A0SBS120): OVER RUN REVERSE
"A0_FCORA"	I 259.1	BOOL	// (A0SBS120): OVER RUN FORWARD
"A0_DI10"	I 259.2	BOOL	// (A0SBS120): DIGITAL INPUT 10
"A0_DI11"	I 259.3	BOOL	// (A0SBS120): DIGITAL INPUT 11
"Z1SPA2CFP"	I 295.0	BOOL	// (Z1SPA2.SI1): CONTROL CERRAMIENTO PUERTA
"A0_POW_I"	I 312.0	BOOL	// (A0SBS120):DRIVE POWER
"A0_SS1_I"	I 312.1	BOOL	// (A0SBS120):SS1 DRIVE OK
"A0_SS2_1"	I 312.2	BOOL	// (A0SBS120):SS2 DRIVE OK
"A0_SOS_I"	I 312.3	BOOL	// (A0SBS120):SOS DRIVE OK
"A0_SLS_I"	I 312.4	BOOL	// (A0SBS120):SLS DRIVE OK
"A0_INT_I"	I 312.7	BOOL	// (A0SBS120):DRIVE INT EV
"A0_L1SLS_I"	I 313.1	BOOL	// (A0SBS120):SLS LIMIT 1 SELECTION
"A0_L2SLS_I"	I 313.2	BOOL	// (A0SBS120):SLS LIMIT 2 SELECTION
"Z1SPA1BMCY"	I 350.7	BOOL	// (Z1SPA1.I0): BOTON FUNCIONAMIENTO DE CICLO
"Z1SPA1BDACY"	I 351.0	BOOL	// (Z1SPA1.I1): BOTON DENANDA PARADA CICLO
"Z1SPA1SPES"	I 351.3	BOOL	// (Z1SPA1.I1): SWITCH ON / OFF PORTÃO
"Z1SPA1SS"	I 353.7	BOOL	// (Z1SPA1.SI0): SELECTOR DE SEGURIDAD
"Z1SPA1CFP"	I 354.0	BOOL	// (Z1SPA1.SI1): CONTROL CERRAMIENTO PUERTA
"Z2CCAU"	I 400.0	BOOL	// (Z2ZB.M02): CONTROL RETORNO COMUN SEGURIDAD AU
"Z2CCES"	I 400.1	BOOL	// (Z2ZB.M02): CONTROL RETORNO COMUN SEGURIDAD ES
"Z2CCFZ"	I 400.2	BOOL	// (Z2ZB.M02): CONTROL RETORNO COMUN SEGURIDAD FZ
"Z2CCRL"	I 400.3	BOOL	// (Z2ZB.M02): CONTROL RETORNO COMUN SEGURIDAD RL
"Z2CCB24Z"	I 400.4	BOOL	// (Z2ZB.M02): RETORNO CONTROL DISJUNTOR 24V (24Z)
"Z2CCB24R"	I 400.5	BOOL	// (Z2ZB.M02): RETORNO CONTROL DISJUNTOR 24V (24R)
"Z2CCB24SC"	I 400.6	BOOL	// (Z2ZB.M02): RETORNO CONTROL DISJUNTOR 24V (SC)
"B0DPG1"	I 400.7	BOOL	// (Z2ZB.M02): Detector Presencia de Griper 1
"Z2CP7B"	I 401.0	BOOL	// (Z2ZB.M03): CONTROL PRESION 7 BARS
"Z2CRM"	I 401.1	BOOL	// (Z2ZB.M03): RETORNO RELE CONTROL DE MASA
"Z2CCB400_1"	I 401.2	BOOL	// (Z2ZB.M03): Breaker Control 400V (SDB1)
"Z2CRO_11"	I 401.3	BOOL	// (Z2ZB.M03): Safety Contactor Control 1 (SDB1)
"Z2CRO_12"	I 401.4	BOOL	// (Z2ZB.M03): Safety Contactor Control 2 (SDB1)
"Z2CCB400_2"	I 401.5	BOOL	// (Z2ZB.M03): Breaker Control 400V (SDB2)
"Z2CRO_21"	I 401.6	BOOL	// (Z2ZB.M03): Safety Contactor Control 1 (SDB2)
"Z2CRO_22"	I 401.7	BOOL	// (Z2ZB.M03): Safety Contactor Control 2 (SDB2)
"B0OP1VAL"	I 402.0	BOOL	// (Z2ZB.M04): Validacion OP1
"B0OP1BROC"	I 402.1	BOOL	// (Z2ZB.M04): Retorno Origen OP1
"B0DPG2"	I 402.3	BOOL	// (Z2ZB.M04): Detector Presencia de Griper 2
"B0OP2BROC"	I 402.6	BOOL	// (Z2ZB.M04): Retorno Origen OP2
"B0OP2VAL"	I 402.7	BOOL	// (Z2ZB.M04): Validacion OP2
"Z2BMCY"	I 403.0	BOOL	// Z2ZB[M05]: START CYCLE BUTTON  (FROM SOP)
"Z2BMA1"	I 403.1	BOOL	// Z2ZB[M05]: ADVANCE BUTTON (FROM SOP)
"Z2BMR1"	I 403.2	BOOL	// Z2ZB[M05]: RETURN BUTTON (FROM SOP)
"Z2BAU1"	I 405.1	BOOL	// (Z2ZB.M10): PARADA DE EMERGENCIA Z2SOP
"B0SSZ"	I 405.2	BOOL	// (Z2ZB.M10): SELECTOR EN SERVICIO ZONA 2
"B1BAU11"	I 411.0	BOOL	// (Z2ZB.M11): PARADA DE EMERGENCIA OP1
"B2BAU11"	I 411.1	BOOL	// (Z2ZB.M11): PARADA DE EMERGENCIA OP2
"B0EFC11"	I 411.2	BOOL	// (Z2ZB.M11): Presencia Estanteria EGS
"B0EFC21"	I 411.3	BOOL	// (Z2ZB.M11): Presencia Estanteria EGS
"B0BK11"	I 417.0	BOOL	// (Z2ZB.M012): Light Curtain 1 (For Trespassing )
"B0BK21"	I 417.1	BOOL	// (Z2ZB.M012): Light Curtain 2 (For Trespassing )
"B0BK31"	I 417.2	BOOL	// (Z2ZB.M012): Light Curtain 3 (For Trespassing )
"B0BK12"	I 417.4	BOOL	// (Z2ZB.M012): Light Curtain 1 (For Trespassing )
"B0BK22"	I 417.5	BOOL	// (Z2ZB.M012): Light Curtain 2 (For Trespassing )
"B0BK32"	I 417.6	BOOL	// (Z2ZB.M012): Light Curtain 3 (For Trespassing )
"B0CRSC4"	I 423.3	BOOL	// (Z2ZB.M15): RELE COMUN DE SOP
"B0DPP1"	I 450.0	BOOL	// PRES PIEZA 1 [DESCENSO] h4m
"B0DPP2"	I 450.1	BOOL	// PRES PIEZA 2 descenso] k9k
"B0DPP3"	I 450.2	BOOL	// PRES PIEZA 3 [POTE DESCOMPRESION] V2 H4M
"B0DPP4"	I 450.3	BOOL	// PRES PIEZA 4 [GANCHO F4]
"B0DPP5"	I 450.4	BOOL	// PRES PIEZA 5 [TUBO CENTRAL]
"B0DPP6"	I 450.5	BOOL	// PRES PIEZA 6 [SILENCIADOR] V3
"B0DPP7"	I 450.6	BOOL	// PRES PIEZA 7 [GANCHO F7]
"B0DPP8"	I 450.7	BOOL	// PRES PIEZA 8 [SENSOR DE COLA]
"B0DRSR11"	I 452.0	BOOL	// DET POS REC SR11
"B0DASR11"	I 452.1	BOOL	// DET POS AV SR11
"B0DRSR21"	I 452.2	BOOL	// DET POS REC SR21
"B0DASR21"	I 452.3	BOOL	// DET POS AV SR21
"B0DRSR31"	I 452.4	BOOL	// DET POS REC SR31
"B0DASR31"	I 452.5	BOOL	// DET POS AV SR31
"B0DRSR51"	I 452.6	BOOL	// DET POS REC SR51
"B0DASR51"	I 452.7	BOOL	// DET POS AV SR51
"B0DRSR41"	I 453.0	BOOL	// DET POS REC SR41
"B0DASR41"	I 453.1	BOOL	// DET POS AV SR41
"B0DRSR82"	I 453.2	BOOL	// DET POS REC SR82
"B0DASR82"	I 453.3	BOOL	// DET POS AV SR82
"B0DRSR52"	I 453.4	BOOL	// DET POS REC SR52
"B0DASR52"	I 453.5	BOOL	// DET POS AV SR52
"B0DRSR53"	I 453.6	BOOL	// DET POS REC SR53
"B0DASR53"	I 453.7	BOOL	// DET POS AV SR53
"B0DRSR61"	I 454.0	BOOL	// DET POS REC SR61
"B0DASR61"	I 454.1	BOOL	// DET POS AV SR61
"B0DRSR71"	I 454.2	BOOL	// DET POS REC SR71
"B0DASR71"	I 454.3	BOOL	// DET POS AV SR71
"B0DRSR81"	I 454.4	BOOL	// DET POS REC SR81
"B0DASR81"	I 454.5	BOOL	// DET POS AV SR81
"B0DRCL91"	I 454.6	BOOL	// DET POS REC CL91
"B0DACL91"	I 454.7	BOOL	// DET POS AV CL91
"B0DACL101"	I 455.0	BOOL	// DET POS AV CL101
"B0DRCL101"	I 455.1	BOOL	// DET POS REC CL101
"B0DP6BAR"	I 457.7	BOOL	// DET PRES 6 BAR
"Z2SPA1BMCY"	I 490.3	BOOL	// (Z2SPA1.I0): BOTON FUNCIONAMIENTO DE CICLO
"Z2SPA1BDACY"	I 490.4	BOOL	// (Z2SPA1.I1): BOTON FUNCIONAMIENTO DE CICLO
"Z2SPA1SPES"	I 490.7	BOOL	// (Z2SPA1.I1): SWITCH ON / OFF PORTÃO
"Z2SPA1SS"	I 493.7	BOOL	// (Z2SPA1.SI0): SELECTOR DE SEGURIDAD
"Z2SPA1CFP"	I 494.0	BOOL	// (Z2SPA1.SI1): CONTROL CERRAMIENTO PUERTA
"B0DATO1"	IB 907	BYTE
"B0DATO2"	IB 908	BYTE
"B0DATO3"	IB 909	BYTE
"B0DATO4"	IB 910	BYTE
"B0DATO5"	IB 911	BYTE
"B0DATO6"	IB 912	BYTE
"B0DATO7"	IB 913	BYTE
"B0DATO8"	IB 914	BYTE
"B0DATO9"	IB 915	BYTE
"B0DATO10"	IB 916	BYTE
"B0DATO11"	IB 917	BYTE
"B0DATO12"	IB 918	BYTE
"B0SEW_POS_LEIDA"	IW 434	WORD
"BA0"	M 0.0	BOOL	// FACILITY: BIT ALWAYS OFF / ILOT: BIT TOUJOURS A 0
"BA1"	M 0.1	BOOL	// FACILITY: BIT ALWAYS ON / ILOT: BIT TOUJOURS A 1
"BA1LIEN"	M 0.2	BOOL	// FACILITY: BIT ALWAYS ON (LINK IN THE PROGRAMMING NETWORK)
"SHUNT"	M 0.3	BOOL	// BIT FOR BYPASS DURING FACILITY START UP / BIT SHUNT POUR LA MISE AU POINT
"PERSO"	M 0.4	BOOL	// NEED TO PERSONALIZE BY THE PROGRAMMER / EQUATION A PERSONNALISER
"POUB"	M 0.5	BOOL	// DUST BIN BIT / BIT POUBELLE
"SYSFROID"	M 0.7	BOOL	// DETECTING COLD START PLC (OB102) / DETECTION DEMARRAGE A FROID API (OB102)
"ICL080S"	M 1.4	BOOL	// BLINKING INFORMATION / INFORMATION CLIGNOTEMENT
"Shunt_BK3"	M 5.0	BOOL
"shunt_pedales"	M 5.1	BOOL
"GPOS"	M 7.0	BOOL	// Griper en Poscion
"IADF"	M 10.1	BOOL	// FACILITY: FAULT RESET INFORMATION (SAFETY)
"IR"	M 10.2	BOOL	// FACILITY: CONTROL ON INFORMATION (SAFETY)
"Z1DEF_MAJ"	M 11.0	BOOL	// ZONE 1: MAJOR FAULT (SAFETY)
"Z1IADF"	M 11.1	BOOL	// ZONE 1: FAULT RESET INFORMATION (SAFETY)
"Z1IR"	M 11.2	BOOL	// ZONE 1: CONTROL ON INFORMATION (SAFETY)
"Z1IAFJ"	M 11.3	BOOL	// ZONE 1: END OF PRODUCTION STOP INFORMATION (SAFETY)
"Z1MAUTO"	M 11.4	BOOL	// ZONE 1: ZONE IN AUTOMATIC MODE (SAFETY)
"A01POSC"	M 11.5	BOOL	// A01: POSICION CARGA (SAFETY)
"A01POST"	M 11.6	BOOL	// A01: POSICION TRABAJO (SAFETY)
"A02POSC"	M 11.7	BOOL	// A02: POSICION cARGA (SAFETY)
"A02POST"	M 12.0	BOOL	// A02: POSICION TRABAJO (SAFETY)
"Z1MANU"	M 12.1	BOOL
"xcero"	M 19.0	BOOL
"Z2DEF_MAJ"	M 21.0	BOOL	// ZONE 2: MAJOR FAULT (SAFETY)
"Z2IADF"	M 21.1	BOOL	// ZONE 2: FAULT RESET INFORMATION (SAFETY)
"Z2IR"	M 21.2	BOOL	// ZONE 2: CONTROL ON INFORMATION (SAFETY)
"Z2IAFJ"	M 21.3	BOOL	// ZONE 2: END OF PRODUCTION STOP INFORMATION (SAFETY)
"Z2MAUTO"	M 21.4	BOOL	// ZONE 2: ZONE IN AUTOMATIC MODE (SAFETY)
"B01POSC"	M 21.5	BOOL	// B01: POSICION CARGA (SAFETY)
"B01POST"	M 21.6	BOOL	// B01: POSICION TRABAJO (SAFETY)
"B02POSC"	M 21.7	BOOL	// B02: POSICION cARGA (SAFETY)
"B02POST"	M 22.0	BOOL	// B02: POSICION TRABAJO (SAFETY)
"Z3DEF_MAJ"	M 30.0	BOOL	// ZONE 3: MAJOR FAULT (SAFETY)
"Z3IADF"	M 30.1	BOOL	// ZONE 3: FAULT RESET INFORMATION (SAFETY)
"Z3IR"	M 30.2	BOOL	// ZONE 3: CONTROL ON INFORMATION (SAFETY)
"Z3IAFJ"	M 30.3	BOOL	// ZONE 3: END OF PRODUCTION STOP INFORMATION (SAFETY)
"Z3MAUTO"	M 30.4	BOOL	// ZONE 3: ZONE IN AUTOMATIC MODE (SAFETY)
"C01POSC"	M 31.0	BOOL	// C01: POSICION CARGA (SAFETY)
"C01POST"	M 31.1	BOOL	// C01: POSICION TRABAJO (SAFETY)
"C02POSC"	M 31.2	BOOL	// C02: POSICION cARGA (SAFETY)
"C02POST"	M 31.3	BOOL	// C02: POSICION TRABAJO (SAFETY)
"C03POSC"	M 31.4	BOOL	// C03: POSICION cARGA (SAFETY)
"C03POST"	M 31.5	BOOL	// C03: POSICION TRABAJO (SAFETY)
"OP2INHIB"	M 40.0	BOOL	// OPERADOR 2 DESABILITADO
"OP1INHIB"	M 40.1	BOOL	// OPERADOR 1 DESABILITADO
"MOP_DROC"	M 40.5	BOOL	// MOP: Retorno a Orijen
"1OPERADOR"	M 40.6	BOOL	// TRABAJA SOLO 1 OPERADOR
"A0SR9_IA"	M 40.7	BOOL	// INFORMACION DEL GRIPO SR9 AVANZADO
"HCB"	M 41.0	BOOL	// Habilitar codigo de barras
"B0_M_LOG_1"	M 50.0	BOOL	// MARCA LOGICA 1
"B01OPERADOR"	M 50.6	BOOL	// TRABAJA SOLO UN OPERADOR
"B0_def_mvt"	M 55.0	BOOL	// DEFECTO DE MOVIMIENTO
"Z2SOP_DROC"	M 60.0	BOOL	// Z2SOP: Demanda Retorno a Orijen
"HCB_X67"	M 120.7	BOOL	// Habilitar codigo de barras X67
"A1CRS"	M 200.2	BOOL	// A1: SAFETY RESET CONDITION / CONDITION DE REARMENENT SECURITE
"A2CRS"	M 200.4	BOOL	// A0: OPERATOR A1 WORK AUTORIZATION / AUTORISATION DE TRAVAIL OPERATEUR A1
"A02_AT_A1"	M 201.0	BOOL	// A02: OPERATOR A1 WORK AUTORIZATION / AUTORISATION DE TRAVAIL OPERATEUR A1
"A02_ET_A1"	M 201.1	BOOL	// A02: OPERATOR A1 WORK COMPLETION / ENREGISTRENENT DE TRAVAIL OPERATEUR A1
"A02_ACTIVA"	M 201.3	BOOL	// A02: CUNA EN PRODUCCION
"B0_AT_B1"	M 300.0	BOOL	// B0: OPERATOR B1 WORK AUTORIZATION / AUTORISATION DE TRAVAIL OPERATEUR B1
"B0_ET_B1"	M 300.1	BOOL	// B1: OPERATOR A1 WORK COMPLETION / ENREGISTRENENT DE TRAVAIL OPERATEUR B1
"B1CRS"	M 300.2	BOOL	// B1: SAFETY RESET CONDITION / CONDITION DE REARMENENT SECURITE
"B01_ACTIVA"	M 300.3	BOOL	// B01: CUNA EN PRODUCCION
"B2CRS"	M 300.4	BOOL	// B0: OPERATOR B1 WORK AUTORIZATION / AUTORISATION DE TRAVAIL OPERATEU
"B02_AT_B1"	M 301.0	BOOL	// B02: OPERATOR A1 WORK AUTORIZATION / AUTORISATION DE TRAVAIL OPERATEUR B1
"B02_ET_B1"	M 301.1	BOOL	// B02: OPERATOR A1 WORK COMPLETION / ENREGISTRENENT DE TRAVAIL OPERATEUR B1
"B1CRSB02"	M 301.2	BOOL	// B2: SAFETY RESET CONDITION / CONDITION DE REARMENENT SECURITE
"B02_ACTIVA"	M 301.3	BOOL	// B02: CUNA EN PRODUCCION
"C0_AT_C1"	M 400.0	BOOL	// C0: OPERATOR A1 WORK AUTORIZATION / AUTORISATION DE TRAVAIL OPERATEUR C1
"C0_ET_C1"	M 400.1	BOOL	// C0: OPERATOR A1 WORK COMPLETION / ENREGISTRENENT DE TRAVAIL OPERATEUR C1
"C1CRSC01"	M 400.2	BOOL	// C1: SAFETY RESET CONDITION / CONDITION DE REARMENENT SECURITE
"C01_ACTIVA"	M 400.3	BOOL	// C01: CUNA EN PRODUCCION
"XA1SFF_MDV"	M 401.0	BOOL	// AUX DE PEDAL PARA MODO DEVERMINAGE
"C1CRSC02"	M 401.2	BOOL	// C1: SAFETY RESET CONDITION / CONDITION DE REARMENENT SECURITE
"C02_ACTIVA"	M 401.3	BOOL	// C02: CUNA EN PRODUCCION
"C1CRSC03"	M 402.2	BOOL	// C1: SAFETY RESET CONDITION / CONDITION DE REARMENENT SECURITE
"C03_ACTIVA"	M 402.3	BOOL	// C03: CUNA EN PRODUCCION
"A0_JOG_AV"	M 500.0	BOOL	// AUTORIZA JOG AVANCO
"A0_JOG_AR"	M 500.1	BOOL	// AUTORIZA JOG RECUO
"REFERENCIA"	M 600.0	BOOL
"JOG_ACTIVE"	M 600.1	BOOL
"XB1SFF_MDV"	M 801.0	BOOL
"A2RC_READY"	M 2200.0	BOOL	// (A2RB.E1): ROBOT PRONTO
"A2MOTORON"	M 2200.1	BOOL	// (A2RB.E1): EN POTENCIA
"A2AUTO"	M 2200.2	BOOL	// (A2RB.E1): COMUTADER EN AUTOMÁTICO
"A2MANU"	M 2200.3	BOOL	// (A2RB.E1): COMUTADER EN MANUAL
"A2REPLI"	M 2200.4	BOOL	// (A2RB.E1): POSICION DE REPLI
"A2RAMVT"	M 2200.7	BOOL	// (A2RB.E1): MOVIMIENTO EN CURSO
"A2HPR"	M 2201.0	BOOL	// (A2RB.E1): FUERA DE PRODUCCION
"A2AOP"	M 2201.1	BOOL	// (A2RB.E1): LLAMADA OPERADOR
"A2DE"	M 2201.2	BOOL	// (A2RB.E1): DERIVADE
"A2TC"	M 2201.3	BOOL	// (A2RB.E1): TOP CICLO
"A2AI"	M 2201.4	BOOL	// (A2RB.E1): PARADA INDUCÃO
"A2APE"	M 2201.5	BOOL	// (A2RB.E1): PARADA PROPIA EXPLORACION
"A2APF"	M 2201.6	BOOL	// (A2RB.E1): PARADA PROPIA FABRICACION
"A2APP"	M 2201.7	BOOL	// (A2RB.E1): PARADA PROPIA PANE
"A2OR1"	M 2202.0	BOOL	// (A2RB.E2): ORDEN 1
"A2OR2"	M 2202.1	BOOL	// (A2RB.E2): ORDEN 2
"A2OR3"	M 2202.2	BOOL	// (A2RB.E2): ORDEN 3
"A2OR4"	M 2202.3	BOOL	// (A2RB.E2): ORDEN 4
"A2OR5"	M 2202.4	BOOL	// (A2RB.E2): ORDEN 5
"A2OR6"	M 2202.5	BOOL	// (A2RB.E2): ORDEN 6
"A2OR7"	M 2202.6	BOOL	// (A2RB.E2): ORDEN 7
"A2OR8"	M 2202.7	BOOL	// (A2RB.E2): ORDEN 8
"A2OR9"	M 2203.0	BOOL	// (A2RB.E2): ORDEN 9
"A2OR10"	M 2203.1	BOOL	// (A2RB.E2): ORDEN 10
"A2OR11"	M 2203.2	BOOL	// (A2RB.E2): ORDEN 11
"A2OR12"	M 2203.3	BOOL	// (A2RB.E2): ORDEN 12
"A2OR13"	M 2203.4	BOOL	// (A2RB.E2): ORDEN 13
"A2OR14"	M 2203.5	BOOL	// (A2RB.E2): ORDEN 14
"A2OR15"	M 2203.6	BOOL	// (A2RB.E2): ORDEN 15
"A2OR16"	M 2203.7	BOOL	// (A2RB.E2): ORDEN 16
"A2CCHDE"	M 2204.0	BOOL	// (A2RB.E3): INFORMACION TROCADER DESTRAVADE
"A2CCHVE"	M 2204.1	BOOL	// (A2RB.E3): INFORMACION TROCADER TRAVADE
"A2CPO"	M 2204.2	BOOL	// (A2RB.E3): SENSOR PRESENCA HERRAMIENTA
"A2CPADV"	M 2204.3	BOOL	// (A2RB.E3): CONTROL PRESION DE AR DESBLOQUIADO
"A2CPAV"	M 2204.4	BOOL	// (A2RB.E3): CONTROL PRESION DE AR BLOQUIADO
"A2CPAS"	M 2204.5	BOOL	// (A2RB.E3): CONTROL DE PRESION DE AR (EV SEGURIDAD)
"A2COHSUP"	M 2204.6	BOOL	// (A2RB.E3): CONTROL HERRAMIENTA FUERA DE SUPORTE
"A2CFRO_ES"	M 2204.7	BOOL	// (A2RB.E3): CONTROL FRO COLOCAR EN SERVICO
"A2CFRO_ZF"	M 2205.0	BOOL	// (A2RB.E3): CONTROL FRO CIERRE ZONE 1
"A2CPAIR"	M 2205.1	BOOL	// (A2RB.E3): CONTROL PRESION AR DE ROBOT
"A2P1KCP"	M 2205.2	BOOL	// (A2RB.E3): KCP ROBOT - PESO 1
"A2P2KCP"	M 2205.3	BOOL	// (A2RB.E3): KCP ROBOT - PESO 2
"A2P4KCP"	M 2205.4	BOOL	// (A2RB.E3): KCP ROBOT - PESO 4
"A2P8KCP"	M 2205.5	BOOL	// (A2RB.E3): KCP ROBOT - PESO 8
"A2P16KCP"	M 2205.6	BOOL	// (A2RB.E3): KCP ROBOT - PESO 16
"A2P32KCP"	M 2205.7	BOOL	// (A2RB.E3): KCP ROBOT - PESO 32
"A2ORO1"	M 2208.0	BOOL	// (A2RB.E5): ORDEN HERRAMIENTA 1
"A2ORO2"	M 2208.1	BOOL	// (A2RB.E5): ORDEN HERRAMIENTA 2
"A2ORO3"	M 2208.2	BOOL	// (A2RB.E5): ORDEN HERRAMIENTA 3
"A2ORO4"	M 2208.3	BOOL	// (A2RB.E5): ORDEN HERRAMIENTA 4
"A2ORO5"	M 2208.4	BOOL	// (A2RB.E5): ORDEN HERRAMIENTA 5
"A2ORO6"	M 2208.5	BOOL	// (A2RB.E5): ORDEN HERRAMIENTA 6
"A2ORO7"	M 2208.6	BOOL	// (A2RB.E5): ORDEN HERRAMIENTA 7
"A2ORO8"	M 2208.7	BOOL	// (A2RB.E5): ORDEN HERRAMIENTA 8
"A2ORO9"	M 2209.0	BOOL	// (A2RB.E5): ORDEN HERRAMIENTA 9
"A2ORO10"	M 2209.1	BOOL	// (A2RB.E5): ORDEN HERRAMIENTA 10
"A2ORO11"	M 2209.2	BOOL	// (A2RB.E5): ORDEN HERRAMIENTA 11
"A2ORO12"	M 2209.3	BOOL	// (A2RB.E5): ORDEN HERRAMIENTA 12
"A2ORO13"	M 2209.4	BOOL	// (A2RB.E5): ORDEN HERRAMIENTA 13
"A2ORO14"	M 2209.5	BOOL	// (A2RB.E5): ORDEN HERRAMIENTA 14
"A2ORO15"	M 2209.6	BOOL	// (A2RB.E5): ORDEN HERRAMIENTA 15
"A2ORO16"	M 2209.7	BOOL	// (A2RB.E5): ORDEN HERRAMIENTA 16
"A2OR17"	M 2214.0	BOOL	// (A2RB.E8): ORDEN 17
"A2OR18"	M 2214.1	BOOL	// (A2RB.E8): ORDEN 18
"A2OR19"	M 2214.2	BOOL	// (A2RB.E8): ORDEN 19
"A2OR20"	M 2214.3	BOOL	// (A2RB.E8): ORDEN 20
"A2OR21"	M 2214.4	BOOL	// (A2RB.E8): ORDEN 21
"A2OR22"	M 2214.5	BOOL	// (A2RB.E8): ORDEN 22
"A2OR23"	M 2214.6	BOOL	// (A2RB.E8): ORDEN 23
"A2OR24"	M 2214.7	BOOL	// (A2RB.E8): ORDEN 24
"A2OR25"	M 2215.0	BOOL	// (A2RB.E8): ORDEN 25
"A2OR26"	M 2215.1	BOOL	// (A2RB.E8): ORDEN 26
"A2OR27"	M 2215.2	BOOL	// (A2RB.E8): ORDEN 27
"A2OR28"	M 2215.3	BOOL	// (A2RB.E8): ORDEN 28
"A2OR29"	M 2215.4	BOOL	// (A2RB.E8): ORDEN 29
"A2OR30"	M 2215.5	BOOL	// (A2RB.E8): ORDEN 30
"A2OR31"	M 2215.6	BOOL	// (A2RB.E8): ORDEN 31
"A2OR32"	M 2215.7	BOOL	// (A2RB.E8): ORDEN 32
"A2AEVRB"	M 2216.0	BOOL	// (A2RB.S1): AUTORIZACION DE EVOLUCION
"A2DMSP"	M 2216.1	BOOL	// (A2RB.S1): SOLICITUD PARA ENERGIZAR
"A2STOP"	M 2216.2	BOOL	// (A2RB.S1): PARADA ROBOT
"A2DDCY"	M 2216.3	BOOL	// (A2RB.S1): INICIO CICLO
"A2DEV"	M 2216.4	BOOL	// (A2RB.S1): DEVERMINAGE
"A2CVC_0"	M 2216.5	BOOL	// (A2RB.S1): CONTROL VALIDACION CODE A 0
"A2CVC_1"	M 2216.6	BOOL	// (A2RB.S1): CONTROL VALIDACION CODE A 1
"A2CPCO"	M 2216.7	BOOL	// (A2RB.S1): CONTOLE CÓDIGO DE PARIDADE
"A2C1"	M 2217.0	BOOL	// (A2RB.S1): CÓDIGO PESO 1
"A2C2"	M 2217.1	BOOL	// (A2RB.S1): CÓDIGO PESO 2
"A2C4"	M 2217.2	BOOL	// (A2RB.S1): CÓDIGO PESO 4
"A2C8"	M 2217.3	BOOL	// (A2RB.S1): CÓDIGO PESO 8
"A2C16"	M 2217.4	BOOL	// (A2RB.S1): CÓDIGO PESO 16
"A2C32"	M 2217.5	BOOL	// (A2RB.S1): CÓDIGO PESO 32
"A2C64"	M 2217.6	BOOL	// (A2RB.S1): CÓDIGO PESO 64
"A2C128"	M 2217.7	BOOL	// (A2RB.S1): CÓDIGO PESO 128
"A2EV1"	M 2218.0	BOOL	// (A2RB.S2): EVENTO 1
"A2EV2"	M 2218.1	BOOL	// (A2RB.S2): EVENTO 2
"A2EV3"	M 2218.2	BOOL	// (A2RB.S2): EVENTO 3
"A2EV4"	M 2218.3	BOOL	// (A2RB.S2): EVENTO 4
"A2EV5"	M 2218.4	BOOL	// (A2RB.S2): EVENTO 5
"A2EV6"	M 2218.5	BOOL	// (A2RB.S2): EVENTO 6
"A2EV7"	M 2218.6	BOOL	// (A2RB.S2): EVENTO 7
"A2EV8"	M 2218.7	BOOL	// (A2RB.S2): EVENTO 8
"A2EV9"	M 2219.0	BOOL	// (A2RB.S2): EVENTO 9
"A2EV10"	M 2219.1	BOOL	// (A2RB.S2): EVENTO 10
"A2EV11"	M 2219.2	BOOL	// (A2RB.S2): EVENTO 11
"A2EV12"	M 2219.3	BOOL	// (A2RB.S2): EVENTO 12
"A2EV13"	M 2219.4	BOOL	// (A2RB.S2): EVENTO 13
"A2EV14"	M 2219.5	BOOL	// (A2RB.S2): EVENTO 14
"A2EV15"	M 2219.6	BOOL	// (A2RB.S2): EVENTO 15
"A2EV16"	M 2219.7	BOOL	// (A2RB.S2): EVENTO 16
"A2ENPRO"	M 2220.0	BOOL	// (A2RB.S3): EN PRODUCCION
"A2RFZ"	M 2220.1	BOOL	// (A2RB.S3): ZONA CERRADA
"A2GS1"	M 2222.0	BOOL	// (A2RB.S4): GRUPO DE SEQUENCIA PESO 1
"A2GS2"	M 2222.1	BOOL	// (A2RB.S4): GRUPO DE SEQUENCIA PESO 2
"A2GS4"	M 2222.2	BOOL	// (A2RB.S4): GRUPO DE SEQUENCIA PESO 4
"A2GS8"	M 2222.3	BOOL	// (A2RB.S4): GRUPO DE SEQUENCIA PESO 8
"A2E1_SRE"	M 2222.4	BOOL	// (A2RB.S4): INFO DETECCION RETROCESOSEQUENCIA 1
"A2E1_SAV"	M 2222.5	BOOL	// (A2RB.S4): INFO DETECCION AVANCE SEQUENCIA 1
"A2E2_SRE"	M 2222.6	BOOL	// (A2RB.S4): INFO DETECCION RETROCESOSEQUENCIA 2
"A2E2_SAV"	M 2222.7	BOOL	// (A2RB.S4): INFO DETECCION AVANCE SEQUENCIA 2
"A2DECH"	M 2223.0	BOOL	// (A2RB.S4): COMANDE DESBLOQUEIO TROCADER
"A2EVO1"	M 2224.0	BOOL	// (A2RB.S5): EVENTO HERRAMIENTA 1
"A2EVO2"	M 2224.1	BOOL	// (A2RB.S5): EVENTO HERRAMIENTA 2
"A2EVO3"	M 2224.2	BOOL	// (A2RB.S5): EVENTO HERRAMIENTA 3
"A2EVO4"	M 2224.3	BOOL	// (A2RB.S5): EVENTO HERRAMIENTA 4
"A2EVO5"	M 2224.4	BOOL	// (A2RB.S5): EVENTO HERRAMIENTA 5
"A2EVO6"	M 2224.5	BOOL	// (A2RB.S5): EVENTO HERRAMIENTA 6
"A2EVO7"	M 2224.6	BOOL	// (A2RB.S5): EVENTO HERRAMIENTA 7
"A2EVO8"	M 2224.7	BOOL	// (A2RB.S5): EVENTO HERRAMIENTA 8
"A2EVO9"	M 2225.0	BOOL	// (A2RB.S5): EVENTO HERRAMIENTA 9
"A2EVO10"	M 2225.1	BOOL	// (A2RB.S5): EVENTO HERRAMIENTA 10
"A2EVO11"	M 2225.2	BOOL	// (A2RB.S5): EVENTO HERRAMIENTA 11
"A2EVO12"	M 2225.3	BOOL	// (A2RB.S5): EVENTO HERRAMIENTA 12
"A2EVO13"	M 2225.4	BOOL	// (A2RB.S5): EVENTO HERRAMIENTA 13
"A2EVO14"	M 2225.5	BOOL	// (A2RB.S5): EVENTO HERRAMIENTA 14
"A2EVO15"	M 2225.6	BOOL	// (A2RB.S5): EVENTO HERRAMIENTA 15
"A2EVO16"	M 2225.7	BOOL	// (A2RB.S5): EVENTO HERRAMIENTA 16
"A2EV17"	M 2230.0	BOOL	// (A2RB.S8): EVENTO 17
"A2EV18"	M 2230.1	BOOL	// (A2RB.S8): EVENTO 18
"A2EV19"	M 2230.2	BOOL	// (A2RB.S8): EVENTO 19
"A2EV20"	M 2230.3	BOOL	// (A2RB.S8): EVENTO 20
"A2EV21"	M 2230.4	BOOL	// (A2RB.S8): EVENTO 21
"A2EV22"	M 2230.5	BOOL	// (A2RB.S8): EVENTO 22
"A2EV23"	M 2230.6	BOOL	// (A2RB.S8): EVENTO 23
"A2EV24"	M 2230.7	BOOL	// (A2RB.S8): EVENTO 24
"A2EV25"	M 2231.0	BOOL	// (A2RB.S8): EVENTO 25
"A2EV26"	M 2231.1	BOOL	// (A2RB.S8): EVENTO 26
"A2EV27"	M 2231.2	BOOL	// (A2RB.S8): EVENTO 27
"A2EV28"	M 2231.3	BOOL	// (A2RB.S8): EVENTO 28
"A2EV29"	M 2231.4	BOOL	// (A2RB.S8): EVENTO 29
"A2EV30"	M 2231.5	BOOL	// (A2RB.S8): EVENTO 30
"A2EV31"	M 2231.6	BOOL	// (A2RB.S8): EVENTO 31
"A2EV32"	M 2231.7	BOOL	// (A2RB.S8): EVENTO 32
"A3RC_READY"	M 2232.0	BOOL	// (A3RB.E1): ROBOT PRONTO
"A3MOTORON"	M 2232.1	BOOL	// (A3RB.E1): EN POTENCIA
"A3AUTO"	M 2232.2	BOOL	// (A3RB.E1): COMUTADER EN AUTOMÁTICO
"A3MANU"	M 2232.3	BOOL	// (A3RB.E1): COMUTADER EN MANUAL
"A3REPLI"	M 2232.4	BOOL	// (A3RB.E1): POSICION DE REPLI
"A3RAMVT"	M 2232.7	BOOL	// (A3RB.E1): MOVIMIENTO EN CURSO
"A3HPR"	M 2233.0	BOOL	// (A3RB.E1): FUERA DE PRODUCCION
"A3AOP"	M 2233.1	BOOL	// (A3RB.E1): LLAMADA OPERADOR
"A3DE"	M 2233.2	BOOL	// (A3RB.E1): DERIVADE
"A3TC"	M 2233.3	BOOL	// (A3RB.E1): TOP CICLO
"A3AI"	M 2233.4	BOOL	// (A3RB.E1): PARADA INDUCÃO
"A3APE"	M 2233.5	BOOL	// (A3RB.E1): PARADA PROPIA EXPLORACION
"A3APF"	M 2233.6	BOOL	// (A3RB.E1): PARADA PROPIA FABRICACION
"A3APP"	M 2233.7	BOOL	// (A3RB.E1): PARADA PROPIA PANE
"A3OR1"	M 2234.0	BOOL	// (A3RB.E2): ORDEN 1
"A3OR2"	M 2234.1	BOOL	// (A3RB.E2): ORDEN 2
"A3OR3"	M 2234.2	BOOL	// (A3RB.E2): ORDEN 3
"A3OR4"	M 2234.3	BOOL	// (A3RB.E2): ORDEN 4
"A3OR5"	M 2234.4	BOOL	// (A3RB.E2): ORDEN 5
"A3OR6"	M 2234.5	BOOL	// (A3RB.E2): ORDEN 6
"A3OR7"	M 2234.6	BOOL	// (A3RB.E2): ORDEN 7
"A3OR8"	M 2234.7	BOOL	// (A3RB.E2): ORDEN 8
"A3OR9"	M 2235.0	BOOL	// (A3RB.E2): ORDEN 9
"A3OR10"	M 2235.1	BOOL	// (A3RB.E2): ORDEN 10
"A3OR11"	M 2235.2	BOOL	// (A3RB.E2): ORDEN 11
"A3OR12"	M 2235.3	BOOL	// (A3RB.E2): ORDEN 12
"A3OR13"	M 2235.4	BOOL	// (A3RB.E2): ORDEN 13
"A3OR14"	M 2235.5	BOOL	// (A3RB.E2): ORDEN 14
"A3OR15"	M 2235.6	BOOL	// (A3RB.E2): ORDEN 15
"A3OR16"	M 2235.7	BOOL	// (A3RB.E2): ORDEN 16
"A3CCHDE"	M 2236.0	BOOL	// (A3RB.E3): INFORMACION TROCADER DESTRAVADE
"A3CCHVE"	M 2236.1	BOOL	// (A3RB.E3): INFORMACION TROCADER TRAVADE
"A3CPO"	M 2236.2	BOOL	// (A3RB.E3): SENSOR PRESENCA HERRAMIENTA
"A3CPADV"	M 2236.3	BOOL	// (A3RB.E3): CONTROL PRESION DE AR DESBLOQUEIO
"A3CPAV"	M 2236.4	BOOL	// (A3RB.E3): CONTROL PRESION DE AR BLOQUEIO
"A3CPAS"	M 2236.5	BOOL	// (A3RB.E3): CONTROL DE PRESION DE AR (EV SEGURIDAD)
"A3COHSUP"	M 2236.6	BOOL	// (A3RB.E3): CONTROL HERRAMIENTA FUERA DE SUPORTE
"A3CFRO_ES"	M 2236.7	BOOL	// (A3RB.E3): CONTROL FRO COLOCAR EN SERVICO
"A3CFRO_ZF"	M 2237.0	BOOL	// (A3RB.E3): CONTROL FRO CIERRE ZONE 1
"A3CPAIR"	M 2237.1	BOOL	// (A3RB.E3): CONTROL PRESION AR DE ROBOT
"A3P1KCP"	M 2237.2	BOOL	// (A3RB.E3): KCP ROBOT - PESO 1
"A3P2KCP"	M 2237.3	BOOL	// (A3RB.E3): KCP ROBOT - PESO 2
"A3P4KCP"	M 2237.4	BOOL	// (A3RB.E3): KCP ROBOT - PESO 4
"A3P8KCP"	M 2237.5	BOOL	// (A3RB.E3): KCP ROBOT - PESO 8
"A3P16KCP"	M 2237.6	BOOL	// (A3RB.E3): KCP ROBOT - PESO 16
"A3P32KCP"	M 2237.7	BOOL	// (A3RB.E3): KCP ROBOT - PESO 32
"A3ORO1"	M 2240.0	BOOL	// (A3RB.E5): ORDEN HERRAMIENTA 1
"A3ORO2"	M 2240.1	BOOL	// (A3RB.E5): ORDEN HERRAMIENTA 2
"A3ORO3"	M 2240.2	BOOL	// (A3RB.E5): ORDEN HERRAMIENTA 3
"A3ORO4"	M 2240.3	BOOL	// (A3RB.E5): ORDEN HERRAMIENTA 4
"A3ORO5"	M 2240.4	BOOL	// (A3RB.E5): ORDEN HERRAMIENTA 5
"A3ORO6"	M 2240.5	BOOL	// (A3RB.E5): ORDEN HERRAMIENTA 6
"A3ORO7"	M 2240.6	BOOL	// (A3RB.E5): ORDEN HERRAMIENTA 7
"A3ORO8"	M 2240.7	BOOL	// (A3RB.E5): ORDEN HERRAMIENTA 8
"A3ORO9"	M 2241.0	BOOL	// (A3RB.E5): ORDEN HERRAMIENTA 9
"A3ORO10"	M 2241.1	BOOL	// (A3RB.E5): ORDEN HERRAMIENTA 10
"A3ORO11"	M 2241.2	BOOL	// (A3RB.E5): ORDEN HERRAMIENTA 11
"A3ORO12"	M 2241.3	BOOL	// (A3RB.E5): ORDEN HERRAMIENTA 12
"A3ORO13"	M 2241.4	BOOL	// (A3RB.E5): ORDEN HERRAMIENTA 13
"A3ORO14"	M 2241.5	BOOL	// (A3RB.E5): ORDEN HERRAMIENTA 14
"A3ORO15"	M 2241.6	BOOL	// (A3RB.E5): ORDEN HERRAMIENTA 15
"A3ORO16"	M 2241.7	BOOL	// (A3RB.E5): ORDEN HERRAMIENTA 16
"A3OR17"	M 2246.0	BOOL	// (A3RB.E8): ORDEN 17
"A3OR18"	M 2246.1	BOOL	// (A3RB.E8): ORDEN 18
"A3OR19"	M 2246.2	BOOL	// (A3RB.E8): ORDEN 19
"A3OR20"	M 2246.3	BOOL	// (A3RB.E8): ORDEN 20
"A3OR21"	M 2246.4	BOOL	// (A3RB.E8): ORDEN 21
"A3OR22"	M 2246.5	BOOL	// (A3RB.E8): ORDEN 22
"A3OR23"	M 2246.6	BOOL	// (A3RB.E8): ORDEN 23
"A3OR24"	M 2246.7	BOOL	// (A3RB.E8): ORDEN 24
"A3OR25"	M 2247.0	BOOL	// (A3RB.E8): ORDEN 25
"A3OR26"	M 2247.1	BOOL	// (A3RB.E8): ORDEN 26
"A3OR27"	M 2247.2	BOOL	// (A3RB.E8): ORDEN 27
"A3OR28"	M 2247.3	BOOL	// (A3RB.E8): ORDEN 28
"A3OR29"	M 2247.4	BOOL	// (A3RB.E8): ORDEN 29
"A3OR30"	M 2247.5	BOOL	// (A3RB.E8): ORDEN 30
"A3OR31"	M 2247.6	BOOL	// (A3RB.E8): ORDEN 31
"A3OR32"	M 2247.7	BOOL	// (A3RB.E8): ORDEN 32
"A3AEVRB"	M 2248.0	BOOL	// (A3RB.S1): AUTORIZACION DE EVOLUCION
"A3DMSP"	M 2248.1	BOOL	// (A3RB.S1): SOLICITUD PARA ENERGIZAR
"A3STOP"	M 2248.2	BOOL	// (A3RB.S1): PARADA ROBOT
"A3DDCY"	M 2248.3	BOOL	// (A3RB.S1): INICIO CICLO
"A3DEV"	M 2248.4	BOOL	// (A3RB.S1): DEVERMINAGE
"A3CVC_0"	M 2248.5	BOOL	// (A3RB.S1): CONTROL VALIDACION CODE A 0
"A3CVC_1"	M 2248.6	BOOL	// (A3RB.S1): CONTROL VALIDACION CODE A 1
"A3CPCO"	M 2248.7	BOOL	// (A3RB.S1): CONTOLE CÓDIGO DE PARIDADE
"A3A3"	M 2249.0	BOOL	// (A3RB.S1): CÓDIGO PESO 1
"A3C2"	M 2249.1	BOOL	// (A3RB.S1): CÓDIGO PESO 2
"A3C4"	M 2249.2	BOOL	// (A3RB.S1): CÓDIGO PESO 4
"A3C8"	M 2249.3	BOOL	// (A3RB.S1): CÓDIGO PESO 8
"A3A36"	M 2249.4	BOOL	// (A3RB.S1): CÓDIGO PESO 16
"A3C32"	M 2249.5	BOOL	// (A3RB.S1): CÓDIGO PESO 32
"A3C64"	M 2249.6	BOOL	// (A3RB.S1): CÓDIGO PESO 64
"A3A328"	M 2249.7	BOOL	// (A3RB.S1): CÓDIGO PESO 128
"A3EV1"	M 2250.0	BOOL	// (A3RB.S2): EVENTO 1
"A3EV2"	M 2250.1	BOOL	// (A3RB.S2): EVENTO 2
"A3EV3"	M 2250.2	BOOL	// (A3RB.S2): EVENTO 3
"A3EV4"	M 2250.3	BOOL	// (A3RB.S2): EVENTO 4
"A3EV5"	M 2250.4	BOOL	// (A3RB.S2): EVENTO 5
"A3EV6"	M 2250.5	BOOL	// (A3RB.S2): EVENTO 6
"A3EV7"	M 2250.6	BOOL	// (A3RB.S2): EVENTO 7
"A3EV8"	M 2250.7	BOOL	// (A3RB.S2): EVENTO 8
"A3EV9"	M 2251.0	BOOL	// (A3RB.S2): EVENTO 9
"A3EV10"	M 2251.1	BOOL	// (A3RB.S2): EVENTO 10
"A3EV11"	M 2251.2	BOOL	// (A3RB.S2): EVENTO 11
"A3EV12"	M 2251.3	BOOL	// (A3RB.S2): EVENTO 12
"A3EV13"	M 2251.4	BOOL	// (A3RB.S2): EVENTO 13
"A3EV14"	M 2251.5	BOOL	// (A3RB.S2): EVENTO 14
"A3EV15"	M 2251.6	BOOL	// (A3RB.S2): EVENTO 15
"A3EV16"	M 2251.7	BOOL	// (A3RB.S2): EVENTO 16
"A3ENPRO"	M 2252.0	BOOL	// (A3RB.S3): EN PRODUCCION
"A3RFZ"	M 2252.1	BOOL	// (A3RB.S3): ZONA CERRADA
"A3GS1"	M 2254.0	BOOL	// (A3RB.S4): GRUPO DE SEQUENCIA PESO 1
"A3GS2"	M 2254.1	BOOL	// (A3RB.S4): GRUPO DE SEQUENCIA PESO 2
"A3GS4"	M 2254.2	BOOL	// (A3RB.S4): GRUPO DE SEQUENCIA PESO 4
"A3GS8"	M 2254.3	BOOL	// (A3RB.S4): GRUPO DE SEQUENCIA PESO 8
"A3E1_SRE"	M 2254.4	BOOL	// (A3RB.S4): INFO DETECCION RETROCESOSEQUENCIA 1
"A3E1_SAV"	M 2254.5	BOOL	// (A3RB.S4): INFO DETECCION AVANCE SEQUENCIA 1
"A3E2_SRE"	M 2254.6	BOOL	// (A3RB.S4): INFO DETECCION RETROCESOSEQUENCIA 2
"A3E2_SAV"	M 2254.7	BOOL	// (A3RB.S4): INFO DETECCION AVANCE SEQUENCIA 2
"A3DECH"	M 2255.0	BOOL	// (A3RB.S4): COMANDE DESBLOQUEIO TROCADER
"A3EVO1"	M 2256.0	BOOL	// (A3RB.S5): EVENTO HERRAMIENTA 1
"A3EVO2"	M 2256.1	BOOL	// (A3RB.S5): EVENTO HERRAMIENTA 2
"A3EVO3"	M 2256.2	BOOL	// (A3RB.S5): EVENTO HERRAMIENTA 3
"A3EVO4"	M 2256.3	BOOL	// (A3RB.S5): EVENTO HERRAMIENTA 4
"A3EVO5"	M 2256.4	BOOL	// (A3RB.S5): EVENTO HERRAMIENTA 5
"A3EVO6"	M 2256.5	BOOL	// (A3RB.S5): EVENTO HERRAMIENTA 6
"A3EVO7"	M 2256.6	BOOL	// (A3RB.S5): EVENTO HERRAMIENTA 7
"A3EVO8"	M 2256.7	BOOL	// (A3RB.S5): EVENTO HERRAMIENTA 8
"A3EVO9"	M 2257.0	BOOL	// (A3RB.S5): EVENTO HERRAMIENTA 9
"A3EVO10"	M 2257.1	BOOL	// (A3RB.S5): EVENTO HERRAMIENTA 10
"A3EVO11"	M 2257.2	BOOL	// (A3RB.S5): EVENTO HERRAMIENTA 11
"A3EVO12"	M 2257.3	BOOL	// (A3RB.S5): EVENTO HERRAMIENTA 12
"A3EVO13"	M 2257.4	BOOL	// (A3RB.S5): EVENTO HERRAMIENTA 13
"A3EVO14"	M 2257.5	BOOL	// (A3RB.S5): EVENTO HERRAMIENTA 14
"A3EVO15"	M 2257.6	BOOL	// (A3RB.S5): EVENTO HERRAMIENTA 15
"A3EVO16"	M 2257.7	BOOL	// (A3RB.S5): EVENTO HERRAMIENTA 16
"A3EV17"	M 2262.0	BOOL	// (A3RB.S8): EVENTO 17
"A3EV18"	M 2262.1	BOOL	// (A3RB.S8): EVENTO 18
"A3EV19"	M 2262.2	BOOL	// (A3RB.S8): EVENTO 19
"A3EV20"	M 2262.3	BOOL	// (A3RB.S8): EVENTO 20
"A3EV21"	M 2262.4	BOOL	// (A3RB.S8): EVENTO 21
"A3EV22"	M 2262.5	BOOL	// (A3RB.S8): EVENTO 22
"A3EV23"	M 2262.6	BOOL	// (A3RB.S8): EVENTO 23
"A3EV24"	M 2262.7	BOOL	// (A3RB.S8): EVENTO 24
"A3EV25"	M 2263.0	BOOL	// (A3RB.S8): EVENTO 25
"A3EV26"	M 2263.1	BOOL	// (A3RB.S8): EVENTO 26
"A3EV27"	M 2263.2	BOOL	// (A3RB.S8): EVENTO 27
"A3EV28"	M 2263.3	BOOL	// (A3RB.S8): EVENTO 28
"A3EV29"	M 2263.4	BOOL	// (A3RB.S8): EVENTO 29
"A3EV30"	M 2263.5	BOOL	// (A3RB.S8): EVENTO 30
"A3EV31"	M 2263.6	BOOL	// (A3RB.S8): EVENTO 31
"A3EV32"	M 2263.7	BOOL	// (A3RB.S8): EVENTO 32
"C2RC_READY"	M 2296.0	BOOL	// (C2RB.E1): ROBOT PRONTO
"C2MOTORON"	M 2296.1	BOOL	// (C2RB.E1): EN POTENCIA
"C2AUTO"	M 2296.2	BOOL	// (C2RB.E1): COMUTADER EN AUTOMÁTICO
"C2MANU"	M 2296.3	BOOL	// (C2RB.E1): COMUTADER EN MANUAL
"C2REPLI"	M 2296.4	BOOL	// (C2RB.E1): POSICION DE REPLI
"C2RAMVT"	M 2296.7	BOOL	// (C2RB.E1): MOVIMIENTO EN CURSO
"C2HPR"	M 2297.0	BOOL	// (C2RB.E1): FUERA DE PRODUCCION
"C2AOP"	M 2297.1	BOOL	// (C2RB.E1): LLAMADA OPERADOR
"C2DE"	M 2297.2	BOOL	// (C2RB.E1): DERIVADE
"C2TC"	M 2297.3	BOOL	// (C2RB.E1): TOP CICLO
"C2AI"	M 2297.4	BOOL	// (C2RB.E1): PARADA INDUCÃO
"C2APE"	M 2297.5	BOOL	// (C2RB.E1): PARADA PROPIA EXPLORACION
"C2APF"	M 2297.6	BOOL	// (C2RB.E1): PARADA PROPIA FABRICACION
"C2APP"	M 2297.7	BOOL	// (C2RB.E1): PARADA PROPIA PANE
"C2OR1"	M 2298.0	BOOL	// (C2RB.E2): ORDEN 1
"C2OR2"	M 2298.1	BOOL	// (C2RB.E2): ORDEN 2
"C2OR3"	M 2298.2	BOOL	// (C2RB.E2): ORDEN 3
"C2OR4"	M 2298.3	BOOL	// (C2RB.E2): ORDEN 4
"C2OR5"	M 2298.4	BOOL	// (C2RB.E2): ORDEN 5
"C2OR6"	M 2298.5	BOOL	// (C2RB.E2): ORDEN 6
"C2OR7"	M 2298.6	BOOL	// (C2RB.E2): ORDEN 7
"C2OR8"	M 2298.7	BOOL	// (C2RB.E2): ORDEN 8
"C2OR9"	M 2299.0	BOOL	// (C2RB.E2): ORDEN 9
"C2OR10"	M 2299.1	BOOL	// (C2RB.E2): ORDEN 10
"C2OR11"	M 2299.2	BOOL	// (C2RB.E2): ORDEN 11
"C2OR12"	M 2299.3	BOOL	// (C2RB.E2): ORDEN 12
"C2OR13"	M 2299.4	BOOL	// (C2RB.E2): ORDEN 13
"C2OR14"	M 2299.5	BOOL	// (C2RB.E2): ORDEN 14
"C2OR15"	M 2299.6	BOOL	// (C2RB.E2): ORDEN 15
"C2OR16"	M 2299.7	BOOL	// (C2RB.E2): ORDEN 16
"C2CCHDE"	M 2300.0	BOOL	// (C2RB.E3): INFORMACION TROCADER DESTRAVADE
"C2CCHVE"	M 2300.1	BOOL	// (C2RB.E3): INFORMACION TROCADER TRAVADE
"C2CPO"	M 2300.2	BOOL	// (C2RB.E3): SENSOR PRESENCA HERRAMIENTA
"C2CPADV"	M 2300.3	BOOL	// (C2RB.E3): CONTROL PRESION DE AR DESBLOQUEIO
"C2CPAV"	M 2300.4	BOOL	// (C2RB.E3): CONTROL PRESION DE AR BLOQUEIO
"C2CPAS"	M 2300.5	BOOL	// (C2RB.E3): CONTROL DE PRESION DE AR (EV SEGURIDAD)
"C2COHSUP"	M 2300.6	BOOL	// (C2RB.E3): CONTROL HERRAMIENTA FUERA DE SUPORTE
"C2CFRO_ES"	M 2300.7	BOOL	// (C2RB.E3): CONTROL FRO COLOCAR EN SERVICO
"C2CFRO_ZF"	M 2301.0	BOOL	// (C2RB.E3): CONTROL FRO CIERRE ZONE 1
"C2CPAIR"	M 2301.1	BOOL	// (C2RB.E3): CONTROL PRESION AR DE ROBOT
"C2P1KCP"	M 2301.2	BOOL	// (C2RB.E3): KCP ROBOT - PESO 1
"C2P2KCP"	M 2301.3	BOOL	// (C2RB.E3): KCP ROBOT - PESO 2
"C2P4KCP"	M 2301.4	BOOL	// (C2RB.E3): KCP ROBOT - PESO 4
"C2P8KCP"	M 2301.5	BOOL	// (C2RB.E3): KCP ROBOT - PESO 8
"C2P16KCP"	M 2301.6	BOOL	// (C2RB.E3): KCP ROBOT - PESO 16
"C2P32KCP"	M 2301.7	BOOL	// (C2RB.E3): KCP ROBOT - PESO 32
"C2ORO1"	M 2304.0	BOOL	// (C2RB.E5): ORDEN HERRAMIENTA 1
"C2ORO2"	M 2304.1	BOOL	// (C2RB.E5): ORDEN HERRAMIENTA 2
"C2ORO3"	M 2304.2	BOOL	// (C2RB.E5): ORDEN HERRAMIENTA 3
"C2ORO4"	M 2304.3	BOOL	// (C2RB.E5): ORDEN HERRAMIENTA 4
"C2ORO5"	M 2304.4	BOOL	// (C2RB.E5): ORDEN HERRAMIENTA 5
"C2ORO6"	M 2304.5	BOOL	// (C2RB.E5): ORDEN HERRAMIENTA 6
"C2ORO7"	M 2304.6	BOOL	// (C2RB.E5): ORDEN HERRAMIENTA 7
"C2ORO8"	M 2304.7	BOOL	// (C2RB.E5): ORDEN HERRAMIENTA 8
"C2ORO9"	M 2305.0	BOOL	// (C2RB.E5): ORDEN HERRAMIENTA 9
"C2ORO10"	M 2305.1	BOOL	// (C2RB.E5): ORDEN HERRAMIENTA 10
"C2ORO11"	M 2305.2	BOOL	// (C2RB.E5): ORDEN HERRAMIENTA 11
"C2ORO12"	M 2305.3	BOOL	// (C2RB.E5): ORDEN HERRAMIENTA 12
"C2ORO13"	M 2305.4	BOOL	// (C2RB.E5): ORDEN HERRAMIENTA 13
"C2ORO14"	M 2305.5	BOOL	// (C2RB.E5): ORDEN HERRAMIENTA 14
"C2ORO15"	M 2305.6	BOOL	// (C2RB.E5): ORDEN HERRAMIENTA 15
"C2ORO16"	M 2305.7	BOOL	// (C2RB.E5): ORDEN HERRAMIENTA 16
"C2OR17"	M 2310.0	BOOL	// (C2RB.E8): ORDEN 17
"C2OR18"	M 2310.1	BOOL	// (C2RB.E8): ORDEN 18
"C2OR19"	M 2310.2	BOOL	// (C2RB.E8): ORDEN 19
"C2OR20"	M 2310.3	BOOL	// (C2RB.E8): ORDEN 20
"C2OR21"	M 2310.4	BOOL	// (C2RB.E8): ORDEN 21
"C2OR22"	M 2310.5	BOOL	// (C2RB.E8): ORDEN 22
"C2OR23"	M 2310.6	BOOL	// (C2RB.E8): ORDEN 23
"C2OR24"	M 2310.7	BOOL	// (C2RB.E8): ORDEN 24
"C2OR25"	M 2311.0	BOOL	// (C2RB.E8): ORDEN 25
"C2OR26"	M 2311.1	BOOL	// (C2RB.E8): ORDEN 26
"C2OR27"	M 2311.2	BOOL	// (C2RB.E8): ORDEN 27
"C2OR28"	M 2311.3	BOOL	// (C2RB.E8): ORDEN 28
"C2OR29"	M 2311.4	BOOL	// (C2RB.E8): ORDEN 29
"C2OR30"	M 2311.5	BOOL	// (C2RB.E8): ORDEN 30
"C2OR31"	M 2311.6	BOOL	// (C2RB.E8): ORDEN 31
"C2OR32"	M 2311.7	BOOL	// (C2RB.E8): ORDEN 32
"C2AEVRB"	M 2312.0	BOOL	// (C2RB.S1): AUTORIZACION DE EVOLUCION
"C2DMSP"	M 2312.1	BOOL	// (C2RB.S1): SOLICITUD PARA ENERGIZAR
"C2STOP"	M 2312.2	BOOL	// (C2RB.S1): PARADA ROBOT
"C2DDCY"	M 2312.3	BOOL	// (C2RB.S1): INICIO CICLO
"C2DEV"	M 2312.4	BOOL	// (C2RB.S1): DEVERMINAGE
"C2CVC_0"	M 2312.5	BOOL	// (C2RB.S1): CONTROL VALIDACION CODE A 0
"C2CVC_1"	M 2312.6	BOOL	// (C2RB.S1): CONTROL VALIDACION CODE A 1
"C2CPCO"	M 2312.7	BOOL	// (C2RB.S1): CONTOLE CÓDIGO DE PARIDADE
"C2C1"	M 2313.0	BOOL	// (C2RB.S1): CÓDIGO PESO 1
"C2C2"	M 2313.1	BOOL	// (C2RB.S1): CÓDIGO PESO 2
"C2C4"	M 2313.2	BOOL	// (C2RB.S1): CÓDIGO PESO 4
"C2C8"	M 2313.3	BOOL	// (C2RB.S1): CÓDIGO PESO 8
"C2C16"	M 2313.4	BOOL	// (C2RB.S1): CÓDIGO PESO 16
"C2C22"	M 2313.5	BOOL	// (C2RB.S1): CÓDIGO PESO 32
"C2C64"	M 2313.6	BOOL	// (C2RB.S1): CÓDIGO PESO 64
"C2C128"	M 2313.7	BOOL	// (C2RB.S1): CÓDIGO PESO 128
"C2EV1"	M 2314.0	BOOL	// (C2RB.S2): EVENTO 1
"C2EV2"	M 2314.1	BOOL	// (C2RB.S2): EVENTO 2
"C2EV3"	M 2314.2	BOOL	// (C2RB.S2): EVENTO 3
"C2EV4"	M 2314.3	BOOL	// (C2RB.S2): EVENTO 4
"C2EV5"	M 2314.4	BOOL	// (C2RB.S2): EVENTO 5
"C2EV6"	M 2314.5	BOOL	// (C2RB.S2): EVENTO 6
"C2EV7"	M 2314.6	BOOL	// (C2RB.S2): EVENTO 7
"C2EV8"	M 2314.7	BOOL	// (C2RB.S2): EVENTO 8
"C2EV9"	M 2315.0	BOOL	// (C2RB.S2): EVENTO 9
"C2EV10"	M 2315.1	BOOL	// (C2RB.S2): EVENTO 10
"C2EV11"	M 2315.2	BOOL	// (C2RB.S2): EVENTO 11
"C2EV12"	M 2315.3	BOOL	// (C2RB.S2): EVENTO 12
"C2EV13"	M 2315.4	BOOL	// (C2RB.S2): EVENTO 13
"C2EV14"	M 2315.5	BOOL	// (C2RB.S2): EVENTO 14
"C2EV15"	M 2315.6	BOOL	// (C2RB.S2): EVENTO 15
"C2EV16"	M 2315.7	BOOL	// (C2RB.S2): EVENTO 16
"C2ENPRO"	M 2316.0	BOOL	// (C2RB.S3): EN PRODUCCION
"C2RFZ"	M 2316.1	BOOL	// (C2RB.S3): ZONA CERRADA
